// oscat_basic/POUs/List Processing/LIST_NEXT
FUNCTION_BLOCK LIST_NEXT
VAR_INPUT
	SEP : BYTE;
	RST : BOOL;
END_VAR
VAR_IN_OUT
	LIST : STRING(LIST_LENGTH);
END_VAR
VAR_OUTPUT
	LEL : STRING(LIST_LENGTH);
	NUL : BOOL;
END_VAR
VAR
	pos : INT := 1;
	pt : POINTER TO ARRAY[1..LIST_LENGTH] OF BYTE;
	po : POINTER TO ARRAY[1..LIST_LENGTH] OF BYTE;
	c: BYTE;
	write: INT;
END_VAR


(*
version 2.0	21. mar. 2011
programmer 	hugo
tested by		oscat

LIST_NEXT retrieves the next element of a list, starting from element 1 after reset or first init.
when the end of the lisat is reached a '' empty string is returned and NUL is set to true.
die liste liegt als string von elementen vor die mit den zeichen SEP am anfang markiert sind.

*)

pt := ADR(LIST);
po := ADR(LEL);

IF rst THEN
	pos := 1;
END_IF;

IF pt^[pos] = 0 OR pos = LIST_LENGTH THEN
	LEL := '';
	NUL := TRUE;
ELSE
	NUL := FALSE;
	write := 1;
	FOR pos := pos + 1 TO LIST_LENGTH DO
		c := pt^[pos];
		IF c = 0 OR c = SEP THEN
			po^[write] := 0;
			RETURN;
		ELSE
			po^[write] := pt^[pos];
			write := write + 1;
		END_IF;
	END_FOR;
END_IF;




(* revision histroy
hm	25. jun. 2008	rev 1.0
	original release

hm	19. jan. 2011	rev 1.1
	changed string(255) to string(LIST_LENGTH)	

hm	21. mar. 2011	rev 2.0
	all elements start with SEP

*)

END_FUNCTION_BLOCK

// oscat_basic/POUs/List Processing/LIST_RETRIEVE
FUNCTION LIST_RETRIEVE : STRING(LIST_LENGTH)
VAR_INPUT
	SEP : BYTE;
	POS : INT;
END_VAR

VAR
	i :	INT;
	o : INT := 1;
	w : INT := 1;
	pt : POINTER TO ARRAY[1..LIST_LENGTH] OF BYTE;
	po : POINTER TO ARRAY[1..LIST_LENGTH] OF BYTE;
	cnt: INT := 0;
	c: BYTE;
END_VAR


(*
version 2.0		21. mar. 2011
programmer 	hugo
tested by		oscat

LIST_RETRIEVE liefert das element an der stelle pos einer liste und löscht das element aus der liste.
die liste liegt als string von elementen vor die mit den zeichen SEP separiert sind.

*)
(*All VAR_IN_OUT variables have been moved to the end of the declaration due to compatibility reasons*)
VAR_IN_OUT
	LIST : STRING(LIST_LENGTH);
END_VAR

(* load pointers *)
pt := ADR(LIST);
po := ADR(LIST_RETRIEVE);

IF pos > 0 THEN
	FOR i := 1 TO LIST_LENGTH DO
		c := pt^[i];
		IF c = 0 THEN
			po^[o] := 0;
			IF cnt < pos THEN pt^[w + 1] := 0; ELSE pt^[w] := 0; END_IF;
			RETURN;
		ELSIF cnt = pos AND c <> SEP THEN				(* we have found the element *)
			po^[o] := pt^[i];
			o := o + 1;
		ELSIF cnt >= pos THEN
			pt^[w] := c;
			w := w + 1;
		ELSE
			w := i;
		END_IF;
		IF c = sep THEN cnt := cnt + 1; END_IF;
	END_FOR;
ELSE
	LIST_RETRIEVE := '';
END_IF;


(* revision histroy
hm	28. jun. 2008	rev 1.0
	original release

hm	19. jan. 2011	rev 1.1
	changed string(255) to string(LIST_LENGTH)

hm	21. mar. 2011	rev 2.0
	all elements start with SEP
*)

END_FUNCTION

// oscat_basic/POUs/List Processing/LIST_RETRIEVE_LAST
FUNCTION LIST_RETRIEVE_LAST : STRING(LIST_LENGTH)
VAR_INPUT
	SEP : BYTE;
END_VAR

VAR
	i :	INT;
	last : INT := 1;
	pt : POINTER TO ARRAY[1..LIST_LENGTH] OF BYTE;
	c: BYTE;
END_VAR


(*
version 2.0		21. mar. 2011
programmer 	hugo
tested by		oscat

LIST_RETRIEVE_LAST liefert das letzte element einer liste und löscht das element aus der liste.
die liste liegt als string von elementen vor die mit den zeichen SEP beginnen.

*)
(*All VAR_IN_OUT variables have been moved to the end of the declaration due to compatibility reasons*)
VAR_IN_OUT
	LIST : STRING(LIST_LENGTH);
END_VAR

(* load pointers *)
pt := ADR(LIST);

(* search position of last element *)
FOR i := 1 TO LIST_LENGTH DO
	c := pt^[i];
	IF c = 0 THEN
		EXIT;
	ELSIF C = SEP THEN
		last := i;
	END_IF;
END_FOR;
(* return last element of list *)
LIST_RETRIEVE_LAST := MID(LIST, LIST_LENGTH, last + 1);
(* terminate list at i *)
pt^[last] := 0;



(* revision histroy
hm	21. mar. 2011	rev 2.0
	new module
*)

END_FUNCTION

// oscat_basic/POUs/Logic/FF edge triggered/COUNT_BR
FUNCTION_BLOCK COUNT_BR
VAR_INPUT
	SET : BOOL;
	IN : BYTE;
	UP : BOOL;
	DN : BOOL;
	STEP : BYTE := 1;
	MX : BYTE := 255;
	RST : BOOL;
END_VAR
VAR_OUTPUT
	CNT : BYTE;
END_VAR
VAR
	last_up: BOOL;
	last_dn: BOOL;
END_VAR

(*
	version 1.0	16 jan 2008
	programmer 	hugo
	tested BY	tobias

Count_BR is a byte counter with independen up and dn inputs. the counter counts from 0 to mx and continues at 0 after is has reached mx
a step input sets the counters stepping width.

*)

IF rst THEN
	cnt := 0;
ELSIF set THEN
	cnt := LIMIT(0,in,mx);
ELSIF up AND NOT last_up THEN
	cnt := INT_TO_BYTE(INC(cnt,step,mx));
ELSIF dn AND NOT last_dn THEN
	cnt := INT_TO_BYTE(inc(cnt,-step,mx));
END_IF;
last_up := up;
last_dn := dn;

(* revision history
hm	16. jan 2008	rev 1.0
	original version

*)

END_FUNCTION_BLOCK

// oscat_basic/POUs/Logic/FF edge triggered/COUNT_DR
FUNCTION_BLOCK COUNT_DR
VAR_INPUT
	SET : BOOL;
	IN : DWORD;
	UP : BOOL;
	DN : BOOL;
	STEP : DWORD := 1;
	MX : DWORD := 16#FFFFFFFF;
	RST : BOOL;
END_VAR
VAR_OUTPUT
	CNT : DWORD;
END_VAR
VAR
	last_up: BOOL;
	last_dn: BOOL;
END_VAR

(*
	version 1.1	20. jan. 2011
	programmer 	hugo
	tested BY		tobias

Count_DR is a DWORD counter with independen up and dn inputs. the counter counts from 0 to mx and continues at 0 after is has reached mx
a step input sets the counters stepping width.

*)

IF rst THEN
	cnt := 0;
ELSIF set THEN
	cnt := LIMIT(0,in,mx);
ELSIF up AND NOT last_up THEN
	IF STEP > MX - CNT THEN
		CNT := CNT - MX + STEP - 1;
	ELSE
		CNT := CNT + STEP;
	END_IF;
ELSIF dn AND NOT last_dn THEN
	IF STEP > CNT THEN
		CNT := CNT - STEP + MX + 1;
	ELSE
		CNT := CNT - STEP;
	END_IF;
END_IF;
last_up := up;
last_dn := dn;

(* revision history
hm	12. jun 2008	rev 1.0
	original version

hm	20. jan. 2011	rev 1.1
	corrected init value of MX to 16#FFFFFFFF

*)

END_FUNCTION_BLOCK

// oscat_basic/POUs/Logic/FF edge triggered/FF_D2E
FUNCTION_BLOCK FF_D2E
VAR_INPUT
	D0 : BOOL;
	D1 : BOOL;
	CLK : BOOL;
	RST : BOOL;
END_VAR
VAR_OUTPUT
	Q0 : BOOL;
	Q1 : BOOL;
END_VAR
VAR
	edge : BOOL;
END_VAR

(*
version 1.3	14. mar. 2009
programmer 	hugo
tested by		oscat

dual D-type flip flop with reset and rising clock trigger

*)

IF rst THEN
	Q0 := FALSE;
	Q1 := FALSE;
ELSIF clk AND NOT edge THEN
	Q0 := D0;
	Q1 := D1;
END_IF;
edge := CLK;

(* revision history
hm	25. dec 2007	rev 1.0
	original version

hm	27. dec 2007	rev 1.1
	changed code for better performance

hm	30. oct. 200	rev 1.2
	deleted unnecessary init with 0

hm	14. mar. 2009	rev 1.3
	removed double assignments

*)

END_FUNCTION_BLOCK

// oscat_basic/POUs/Logic/FF edge triggered/FF_D4E
FUNCTION_BLOCK FF_D4E
VAR_INPUT
	D0 : BOOL;
	D1 : BOOL;
	D2 : BOOL;
	D3 : BOOL;
	CLK : BOOL;
	RST : BOOL;
END_VAR
VAR_OUTPUT
	Q0 : BOOL;
	Q1 : BOOL;
	Q2 : BOOL;
	Q3 : BOOL;
END_VAR
VAR
	edge : BOOL;
END_VAR


(*
version 1.3	14. mar. 2009
programmer 	hugo
tested by		oscat

quad D-type flip flop with reset and rising clock trigger

*)

IF rst THEN
	Q0 := FALSE;
	Q1 := FALSE;
	Q2 := FALSE;
	Q3 := FALSE;
ELSIF clk AND NOT edge THEN
	Q0 := D0;
	Q1 := D1;
	Q2 := D2;
	Q3 := D3;
END_IF;
edge := CLK;

(* revision history
hm	4. aug 2006	rev 1.0
	original version

hm	27. dec 2007	rev 1.1
	changed code for better performance

hm	30. oct. 200	rev 1.2
	deleted unnecessary init with 0

hm	14. mar. 2009	rev 1.3
	removed double assignments

*)

END_FUNCTION_BLOCK

// oscat_basic/POUs/Logic/FF edge triggered/FF_DRE
FUNCTION_BLOCK FF_DRE
VAR_INPUT
	SET : BOOL;
	D : BOOL;
	CLK : BOOL;
	RST : BOOL;
END_VAR
VAR_OUTPUT
	Q : BOOL;
END_VAR
VAR
	edge : BOOL;
END_VAR


(*
version 1.2	30. oct. 2008
programmer 	hugo
tested by	oscat

D-type flip flop with set, reset and rising clock trigger

*)

IF rst OR set THEN
	Q := NOT rst;
ELSIF clk AND NOT edge THEN
	Q := D;
END_IF;
edge := CLK;

(* revision history
hm	4. aug 2006		rev 1.0
	original version

hm	27. dec 2007	rev 1.1
	changed code for better performance

hm	30. oct. 2008	rev 1.2
	optimized performance
*)

END_FUNCTION_BLOCK

// oscat_basic/POUs/Logic/FF edge triggered/FF_JKE
FUNCTION_BLOCK FF_JKE
VAR_INPUT
	SET : BOOL;
	J : BOOL;
	CLK : BOOL;
	K : BOOL;
	RST : BOOL;
END_VAR
VAR_OUTPUT
	Q : BOOL;
END_VAR
VAR
	edge : BOOL;
END_VAR


(*
version 1.2	30. oct. 2008
programmer 	hugo
tested by	oscat

JK-type flip flop with set, reset and rising clock trigger
set and reset are asynchron while the FF is rising edge triggered
J=0 and K=0 and CLK >>> no action
J=1 and K=0 and CLK >>> output = 1
J=0 and K=1 and CLK >>> output = 0
J=1 and K=1 and CLK >>> toggle output


*)

IF rst OR set THEN
	Q := NOT rst;
ELSIF clk AND NOT edge THEN
	IF J XOR K THEN Q := J;
	ELSE Q := K XOR Q;
	END_IF;
END_IF;
edge := CLK;

(* revision history
hm	4. aug 2006		rev 1.0
	original version

hm	27. dec 2007	rev 1.1
	changed code for better performance

hm	30. oct. 2008	rev 1.2
	optimized performance
*)

END_FUNCTION_BLOCK

// oscat_basic/POUs/Logic/FF edge triggered/FF_RSE
FUNCTION_BLOCK FF_RSE
VAR_INPUT
	CS : BOOL;
	CR : BOOL;
	RST : BOOL;
END_VAR
VAR_OUTPUT
	Q : BOOL;
END_VAR
VAR
	es, er : BOOL;
END_VAR

(*
version 1.0	16. jul. 2008
programmer 	hugo
tested by	oscat

this is a rising edge triggered rs flip flop
a rising edge on CS sets Q = TRUE and a rising edge on CR sets Q = FALSE.
CR has priority over CS.

*)

IF rst THEN
	(* asynchronous reset *)
	Q := FALSE;
ELSIF CR AND NOT er THEN
	(* rising edge on CR *)
	Q := FALSE;
ELSIF CS AND NOT es THEN
	(* rising edge on CS *)
	Q := TRUE;
END_IF;

es := CS;
er := CR;

(* revision history

hm	16. jul. 2008	rev 1.0
	original version

*)

END_FUNCTION_BLOCK

// oscat_basic/POUs/Logic/FF edge triggered/SELECT_8
FUNCTION_BLOCK SELECT_8
VAR_INPUT
	E : BOOL;
	SET : BOOL;
	IN : BYTE;
	UP : BOOL;
	DN : BOOL;
	RST : BOOL;
END_VAR
VAR_OUTPUT
	Q0, Q1, Q2, Q3, Q4, Q5, Q6, Q7 : BOOL;
	STATE : INT;
END_VAR
VAR
	last_up: BOOL;
	last_dn : BOOL;
END_VAR

(*
	version 1.1	27. feb. 2009
	programmer 	hugo
	tested BY		oscat

select_8 selects one of 8 outputs at any time. the outputscan be selected by up or down keys and an independent anable switches all outouts off if set false


*)

IF rst THEN
	state := 0;
ELSIF set THEN
	state := IN;
ELSIF up AND NOT last_up THEN
	state := inc(state,1,7);
ELSIF dn AND NOT last_dn THEN
	state := inc(state,-1,7);
END_IF;
last_UP := UP;
last_DN := DN;

Q0 := FALSE;
Q1 := FALSE;
Q2 := FALSE;
Q3 := FALSE;
Q4 := FALSE;
Q5 := FALSE;
Q6 := FALSE;
Q7 := FALSE;

IF E THEN
	CASE state OF
		0: Q0 := TRUE;
		1: Q1 := TRUE;
		2: Q2 := TRUE;
		3: Q3 := TRUE;
		4: Q4 := TRUE;
		5: Q5 := TRUE;
		6: Q6 := TRUE;
		7: Q7 := TRUE;
	END_CASE;
END_IF;

(* revision history
hm	16. jan 2008	rev 1.0
	original version

hm	27. feb. 2009	rev 1.1
	renamed input en to e
*)

END_FUNCTION_BLOCK

// oscat_basic/POUs/Logic/FF edge triggered/SHR_4E
FUNCTION_BLOCK SHR_4E
VAR_INPUT
	SET : BOOL;
	D0: BOOL;
	CLK: BOOL;
	RST: BOOL;
END_VAR
VAR_OUTPUT
	Q0: BOOL;
	Q1: BOOL;
	Q2: BOOL;
	Q3: BOOL;
END_VAR
VAR
	trig : R_TRIG;
END_VAR

(*
version 1.1	25. oct. 2008
programmer 	hugo
tested by		tobias

4 bit shift register with reset

*)

(* trig.Q signals a rising edge on clk *)
trig(clk := clk);

IF set OR rst THEN
	Q0 := NOT rst;
	Q1 := Q0;
	Q2 := Q0;
	Q3 := Q0;
ELSIF trig.Q THEN
	Q3 := Q2;
	Q2 := Q1;
	Q1 := Q0;
	Q0 := D0;
END_IF;



(* revision history
hm	4. aug. 2006	rev 1.0
	original version

hm	25. oct. 2008	rev 1.1
	optimized code

*)

END_FUNCTION_BLOCK

// oscat_basic/POUs/Logic/FF edge triggered/SHR_4UDE
FUNCTION_BLOCK SHR_4UDE
VAR_INPUT
	SET : BOOL;
	D0: BOOL;
	D3: BOOL;
	CLK: BOOL;
	DN : BOOL;
	RST: BOOL;

END_VAR
VAR_OUTPUT
	Q0: BOOL;
	Q1: BOOL;
	Q2: BOOL;
	Q3: BOOL;
END_VAR
VAR
	trig : R_TRIG;
END_VAR

(*
version 1.2	14. mar. 2009
programmer 	hugo
tested by		tobias

4 bit shift register with reset up / down direction input

*)

(* trig.Q signals a rising edge on clk *)
trig(clk := clk);

IF set OR rst THEN
	Q0 := NOT RST;
	Q1 := Q0;
	Q2 := Q0;
	Q3 := Q0;
ELSIF trig.Q THEN
	IF dn THEN
		Q0 := Q1;
		Q1 := Q2;
		Q2 := Q3;
		Q3 := D3;
	ELSE
		Q3 := Q2;
		Q2 := Q1;
		Q1 := Q0;
		Q0 := D0;
	END_IF;
END_IF;



(* revision history
hm	4. aug. 2006	rev 1.0
	original version

hm	25. oct. 2008	rev 1.1
	optimized code

hm	14. mar. 2009	rev 1.2
	removed double assignments

*)

END_FUNCTION_BLOCK

// oscat_basic/POUs/Logic/FF edge triggered/SHR_8PLE
FUNCTION_BLOCK SHR_8PLE
VAR_INPUT
	Din : BOOL;
	Dload : BYTE;
	CLK: BOOL;
	UP: BOOL :=1;
	load : BOOL;
	RST: BOOL;
END_VAR
VAR_OUTPUT
	DOut: BOOL;
END_VAR
VAR
	edge : BOOL :=1;
	register : BYTE;
END_VAR

(*
version 1.0	4 aug 2006
programmer 	hugo
tested by	oscat

8 bit shift register with reset and parallel load
the register can shift up or down
it also has a serial input.
the Din input is on Bit0 for up shift and on bit 7 for down shift
the Dout output is on Bit7 for up shift and on bit 0 for down shift
paralle clock is performed clock synchron while a shift is performed first and then the register is reloaded


*)

(* flankenerkennung clk wird high und edge war high reset ist nicht aktiv und set ist nicht aktiv *)
IF CLK AND edge AND NOT rst THEN
	edge := FALSE;	(* flanke wurde erkannt und weitere flankenerkennung wird verhindert bis edge wieder true ist *)
	(* hier ist der code für das flankenevent *)
	IF UP THEN						(*shift up *)
		register := SHL(register,1);
		register.0 := Din;
		Dout := register.7;
	ELSE								(* shift down *);
		register := SHR(register,1);
		register.7 := Din;
		Dout := register.0;
	END_IF;
	IF load THEN							(* the byte on Din will be loaded if load = true *)
		register := Dload;
		IF up THEN Dout := register.7; ELSE Dout := register.0; END_IF;
	END_IF;
END_IF;
IF NOT clk THEN edge := TRUE; END_IF;	(* sobald clk wieder low wird warten auf nächste flanke *)
IF rst THEN									(* wenn reset aktiv dann ausgang rücksetzen *)
	register := 0;
	Dout := FALSE;
END_IF;

END_FUNCTION_BLOCK

// oscat_basic/POUs/Logic/FF edge triggered/SHR_8UDE
FUNCTION_BLOCK SHR_8UDE
VAR_INPUT
	SET : BOOL;
	D0: BOOL;
	D7: BOOL;
	CLK: BOOL;
	DN : BOOL;
	RST: BOOL;
END_VAR
VAR_OUTPUT
	Q0: BOOL;
	Q1: BOOL;
	Q2: BOOL;
	Q3: BOOL;
	Q4: BOOL;
	Q5: BOOL;
	Q6: BOOL;
	Q7: BOOL;
END_VAR
VAR
	trig : R_TRIG;
END_VAR

(*
version 1.2	14. mar. 2009
programmer 	hugo
tested by		tobias

8 bit shift register with reset


*)

(* trig.Q signals a rising edge on clk *)
trig(clk := clk);

IF set OR rst THEN
	Q0 := NOT RST;
	Q1 := Q0;
	Q2 := Q0;
	Q3 := Q0;
	Q4 := Q0;
	Q5 := Q0;
	Q6 := Q0;
	Q7 := Q0;
ELSIF trig.Q THEN
	IF dn THEN
		Q0 := Q1;
		Q1 := Q2;
		Q2 := Q3;
		Q3 := Q4;
		Q4 := Q5;
		Q5 := Q6;
		Q6 := Q7;
		Q7 := D7;
	ELSE
		Q7 := Q6;
		Q6 := Q5;
		Q5 := Q4;
		Q4 := Q3;
		Q3 := Q2;
		Q2 := Q1;
		Q1 := Q0;
		Q0 := D0;
	END_IF;
END_IF;



(* revision history
hm	4. aug. 2006	rev 1.0
	original version

hm	25. oct. 2008	rev 1.1
	optimized code

hm	14. mar. 2009	rev 1.2
	removed double assignments

*)

END_FUNCTION_BLOCK

// oscat_basic/POUs/Logic/FF pulse triggered/LTCH
FUNCTION_BLOCK LTCH
VAR_INPUT
	D : BOOL;
	L : BOOL;
	RST : BOOL;
END_VAR
VAR_OUTPUT
	Q : BOOL;
END_VAR


(*
version 1.2	30. oct. 2008
programmer 	hugo
tested by	oscat

Transparent Latch with asynchronous reset


*)

(* as long as L is true, the latch is transparent and and change of D is transferred to Q *)
(* of course only when there is no asynchronous reset *)
IF rst THEN				(* if asynchronous reset then Q=0 *)
	Q := FALSE;
ELSIF L THEN			(* latch is transparent *)
	Q := D;
END_IF;


(* revision history
hm	4. aug 2006		rev 1.0
	original version

hm	27. dec 2007	rev 1.1
	changed code for better performance

hm	30. oct. 2008	rev 1.2
	deleted unnecessary init with 0

*)

END_FUNCTION_BLOCK

// oscat_basic/POUs/Logic/FF pulse triggered/LTCH_4
FUNCTION_BLOCK LTCH_4
VAR_INPUT
	D0 : BOOL;
	D1 : BOOL;
	D2 : BOOL;
	D3 : BOOL;
	L : BOOL;
	RST : BOOL;
END_VAR
VAR_OUTPUT
	Q0 : BOOL;
	Q1 : BOOL;
	Q2 : BOOL;
	Q3 : BOOL;
END_VAR


(*
version 1.3	14. mar. 2009
programmer 	hugo
tested by		oscat

Quad Transparent Latch with asynchronous reset


*)

(* as long as L is true, the latch is transparent and and change of D is transferred to Q *)
(* of course only when there is no asynchronous reset *)
IF rst THEN			(* if asynchronous reset then Q=0 *)
	Q0 := FALSE;
	Q1 := FALSE;
	Q2 := FALSE;
	Q3 := FALSE;
ELSIF L THEN			(* latch is transparent *)
	Q0 := D0;
	Q1 := D1;
	Q2 := D2;
	Q3 := D3;
END_IF;

(* revision history
hm	4. aug 2006	rev 1.0
	original version

hm	27. dec 2007	rev 1.1
	changed code for better performance

hm	30. oct. 2008	rev 1.2
	deleted unnecessary init with 0

hm	14. mar. 2009	rev 1.3
	removed double assignments

*)

END_FUNCTION_BLOCK

// oscat_basic/POUs/Logic/FF pulse triggered/STORE_8
FUNCTION_BLOCK STORE_8
VAR_INPUT
	Set : BOOL;
	D0,D1, D2, D3, D4, D5, D6, D7 : BOOL;
	Clr : BOOL;
	Rst : BOOL;
END_VAR
VAR_OUTPUT
	Q0, Q1, Q2, Q3, Q4, Q5, Q6, Q7 : BOOL;
END_VAR
VAR
	edge: BOOL;
END_VAR

(*
version 1.2	14. mar. 2009
programmer 	hugo
tested by		oscat

Store_4 stores up to 4 boolean inputs until a reset is clearing the outputs.
the respective output is set with a true at the respective input and stays true until a reset is generated.
a set input is used to set all outputs true at the same time, independent of their inputs.
a clear input is used to reset only the lowest priority of the outputs one at a time.
the lowest priority is q3.

*)

IF rst OR set THEN
	q0 := NOT rst;
	q1 := q0;
	q2 := q0;
	q3 := q0;
	q4 := q0;
	q5 := q0;
	q6 := q0;
	q7 := q0;
ELSE
	IF D0 THEN Q0 := TRUE; END_IF;
	IF D1 THEN Q1 := TRUE; END_IF;
	IF D2 THEN Q2 := TRUE; END_IF;
	IF D3 THEN Q3 := TRUE; END_IF;
	IF D4 THEN Q4 := TRUE; END_IF;
	IF D5 THEN Q5 := TRUE; END_IF;
	IF D6 THEN Q6 := TRUE; END_IF;
	IF D7 THEN Q7 := TRUE; END_IF;

	IF clr AND NOT edge THEN
		IF q0 THEN q0 := FALSE;
		ELSIF q1 THEN q1 := FALSE;
		ELSIF q2 THEN q2 := FALSE;
		ELSIF q3 THEN q3 := FALSE;
		ELSIF q4 THEN q4 := FALSE;
		ELSIF q5 THEN q5 := FALSE;
		ELSIF q6 THEN q6 := FALSE;
		ELSE q7 := FALSE;
		END_IF;
	END_IF;
	edge := clr;
END_IF;


(* revision history
hm	25.12.2007	rev 1.0
	original version

hm	30. oct. 2008	rev 1.1
	optimized performance

hm	14. mar. 2009	rev 1.2
	removed double assignments

*)

END_FUNCTION_BLOCK

// oscat_basic/POUs/Logic/gate logic/BCDC_TO_INT
FUNCTION BCDC_TO_INT : INT
VAR_INPUT
	IN : BYTE;
END_VAR


(*
version 1.1 30. jun. 2008
programmer 	hugo
tested by	oscat

this function converts a two digit bcd number into an integer.

*)

BCDC_TO_INT := (in AND 16#0F) + (SHR(in,4) * 10);

(* revision history
hm	13.12.2007	rev 1.0
	original version

hm	30.6.2008	rev 1.1
	changed name BCD_TO_INT to BCDC_TO_INT to avoid collision with util.lib

*)

END_FUNCTION

// oscat_basic/POUs/Logic/gate logic/BIT_LOAD_B
FUNCTION BIT_LOAD_B : BYTE
VAR_INPUT
	IN : BYTE;
	VAL : BOOL;
	POS : INT;
END_VAR
VAR CONSTANT
	dat : BYTE := 1;
END_VAR

(*
version 1.1	16. mar 2008
programmer 	hugo
tested by	tobias

this function loads a bit into a byte at position pos.
 *)

IF VAL THEN
	BIT_LOAD_B := in OR SHL(dat,pos);
ELSE
	BIT_LOAD_B := in AND (NOT SHL(dat,pos));
END_IF;


(* revision history
hm	29. feb 2008	rev 1.0
	original version

hm	16. mar 2008	rev 1.1
	change input bit to val for compatibility reasons
*)

END_FUNCTION

// oscat_basic/POUs/Logic/gate logic/BIT_LOAD_B2
FUNCTION BIT_LOAD_B2 : BYTE
VAR_INPUT
	I : BYTE;
	D : BOOL;
	P : INT;
	N : INT;
END_VAR


(*
version 1.0 18. oct. 2008
programmer 	hugo
tested by	tobias

this function loads N bits of D at pos P in Byte I

*)

IF D THEN
	BIT_LOAD_B2 := ROL(SHR(BYTE#255, 8 - N) OR ROR(i, P), P);
ELSE
	BIT_LOAD_B2 := ROL(SHL(BYTE#255, N) AND ROR(I, P), P);
END_IF;



(* revision history
hm	18. oct. 2008	rev 1.0
	original version


*)

END_FUNCTION

// oscat_basic/POUs/Logic/gate logic/BIT_LOAD_DW
FUNCTION BIT_LOAD_DW : DWORD
VAR_INPUT
	IN : DWORD;
	VAL : BOOL;
	POS : INT;
END_VAR
VAR CONSTANT
	dat : DWORD := 1;
END_VAR

(*
version 1.1	16. mar 2008
programmer 	hugo
tested by	tobias

this function loads a bit into a DWord at position pos.
 *)

IF val THEN
	BIT_LOAD_DW := in OR SHL(dat,pos);
ELSE
	BIT_LOAD_DW := in AND (NOT SHL(dat,pos));
END_IF;


(* revision history
hm	29. feb 2008	rev 1.0
	original version

hm	16. mar 2008	rev 1.1
	change input bit to val for compatibility reasons
*)

END_FUNCTION

// oscat_basic/POUs/Logic/gate logic/BIT_LOAD_DW2
FUNCTION BIT_LOAD_DW2 : DWORD
VAR_INPUT
	I : DWORD;
	D : BOOL;
	P : INT;
	N : INT;
END_VAR


(*
version 1.0 18. oct. 2008
programmer 	hugo
tested by	tobias

this function loads N bits of D at pos P in DWORD I

*)

IF D THEN
	BIT_LOAD_DW2 := ROL(SHR(DWORD#4294967295, 32 - N) OR ROR(i, P), P);
ELSE
	BIT_LOAD_DW2 := ROL(SHL(DWORD#4294967295, N) AND ROR(I, P), P);
END_IF;



(* revision history
hm	18. oct. 2008	rev 1.0
	original version


*)

END_FUNCTION

// oscat_basic/POUs/Logic/gate logic/BIT_LOAD_W
FUNCTION BIT_LOAD_W : WORD
VAR_INPUT
	IN : WORD;
	VAL : BOOL;
	POS : INT;
END_VAR
VAR CONSTANT
	dat : WORD := 1;
END_VAR

(*
version 1.1	16. mar 2008
programmer 	hugo
tested by	tobias

this function loads a bit into a Word at position pos.
 *)

IF val THEN
	BIT_LOAD_W := in OR SHL(dat,pos);
ELSE
	BIT_LOAD_W := in AND (NOT SHL(dat,pos));
END_IF;


(* revision history
hm	29. feb 2008	rev 1.0
	original version

hm	16. mar 2008	rev 1.1
	change input bit to val for compatibility reasons
*)

END_FUNCTION

// oscat_basic/POUs/Logic/gate logic/BIT_LOAD_W2
FUNCTION BIT_LOAD_W2 : WORD
VAR_INPUT
	I : WORD;
	D : BOOL;
	P : INT;
	N : INT;
END_VAR


(*
version 1.0 18. oct. 2008
programmer 	hugo
tested by	tobias

this function loads N bits of D at pos P in WORD I

*)

IF D THEN
	BIT_LOAD_W2 := ROL(SHR(WORD#65535, 16 - N) OR ROR(i, P), P);
ELSE
	BIT_LOAD_W2 := ROL(SHL(WORD#65535, N) AND ROR(I, P), P);
END_IF;



(* revision history
hm	18. oct. 2008	rev 1.0
	original version


*)

END_FUNCTION

// oscat_basic/POUs/Logic/gate logic/BIT_OF_DWORD
FUNCTION BIT_OF_DWORD : BOOL
VAR_INPUT
	in : DWORD;
	N : INT;
END_VAR


(*
version 1.2	6. jun. 2008
programmer 	hugo
tested by	tobias

this function extracts a single bit from the nth position from right (right is lowest bit)
the lowest Bit (Bit0 from in) is selected with N=0.
 *)

BIT_OF_DWORD := (SHR(in,N) AND 16#00000001) > 0;


(* old code used before rev 1.1
temp := SHR(in,n);
Bit_of_Dword := temp.0;
*)


(* revision history
hm	4. aug. 2006	rev 1.0
	original version

hm	29. feb 2008	rev 1.1
	improved performance

hm	6. jun. 2008	rev 1.2
	changes type of input N from byte to int
*)

END_FUNCTION

// oscat_basic/POUs/Logic/gate logic/BIT_TOGGLE_B
FUNCTION BIT_TOGGLE_B : BYTE
VAR_INPUT
	IN : BYTE;
	POS : INT;
END_VAR


(*
version 1.0 18. oct. 2008
programmer 	hugo
tested by	tobias

this function toggles a bit of a BYTE at position pos.

*)

BIT_TOGGLE_B := SHL(BYTE#1, POS) XOR IN;




(* revision history
hm	18. oct. 2008	rev 1.0
	original version


*)

END_FUNCTION

// oscat_basic/POUs/Logic/gate logic/BIT_TOGGLE_DW
FUNCTION BIT_TOGGLE_DW : DWORD
VAR_INPUT
	IN : DWORD;
	POS : INT;
END_VAR


(*
version 1.0 18. oct. 2008
programmer 	hugo
tested by	tobias

this function toggles a bit of a WORD at position pos.

*)

BIT_TOGGLE_DW := SHL(DWORD#1, POS) XOR IN;



(* revision history
hm	18. oct. 2008	rev 1.0
	original version


*)

END_FUNCTION

// oscat_basic/POUs/Logic/gate logic/BIT_TOGGLE_W
FUNCTION BIT_TOGGLE_W : WORD
VAR_INPUT
	IN : WORD;
	POS : INT;
END_VAR


(*
version 1.0 18. oct. 2008
programmer 	hugo
tested by	tobias

this function toggles a bit of a WORD at position pos.

*)

BIT_TOGGLE_W := SHL(WORD#1, POS) XOR IN;



(* revision history
hm	18. oct. 2008	rev 1.0
	original version


*)

END_FUNCTION

// oscat_basic/POUs/Logic/gate logic/BYTE_OF_BIT
FUNCTION BYTE_OF_BIT : BYTE
VAR_INPUT
	B0:BOOL;
	B1:BOOL;
	B2:BOOL;
	B3:BOOL;
	B4:BOOL;
	B5:BOOL;
	B6:BOOL;
	B7:BOOL;
END_VAR


(*
version 1.1	 18. feb 2006
programmer 	hugo
tested by		tobias

this function creates a byte from 8 individual bits

*)

Byte_of_bit := SHL(SHL(SHL(SHL(SHL(SHL(SHL(BOOL_TO_BYTE(B7),1) OR BOOL_TO_BYTE(B6),1) OR BOOL_TO_BYTE(B5),1) OR BOOL_TO_BYTE(B4),1)
	OR BOOL_TO_BYTE(B3),1) OR BOOL_TO_BYTE(B2),1) OR BOOL_TO_BYTE(B1),1) OR BOOL_TO_BYTE(B0);


(* revision history

hm	4. aug 2006		rev 1.0
	original version

hm	18. feb. 2008	rev 1.1
	improved performance

*)

END_FUNCTION

// oscat_basic/POUs/Logic/gate logic/BYTE_OF_DWORD
FUNCTION BYTE_OF_DWORD : BYTE
VAR_INPUT
	in : DWORD;
	N : BYTE;
END_VAR


(*
version 1.2	30. oct. 2008
programmer 	hugo
tested by	oscat

this function extracts a single byte from the nth position from right (right is lowest byte) 
the lower byte (starting with Bit0 from in) is selected with N=0.
*)

BYTE_OF_DWORD := DWORD_TO_BYTE(SHR(in,SHL(n,3)));

(* revision history
hm	17. jan 2007	rev 1.0
	original version

hm	2. jan 2008		rev 1.1
	improved performance

hm	30. oct. 2008	rev 1.2
	improved performance
*)

END_FUNCTION

// oscat_basic/POUs/Logic/gate logic/BYTE_TO_BITS
FUNCTION_BLOCK BYTE_TO_BITS
VAR_INPUT
	IN: BYTE;
END_VAR
VAR_OUTPUT
	B0: BOOL;
	B1: BOOL;
	B2: BOOL;
	B3: BOOL;
	B4: BOOL;
	B5: BOOL;
	B6: BOOL;
	B7: BOOL;
END_VAR


(*
version 1.1	16. mar. 2008
programmer 	hugo
tested by		tobias

this Function Block extracts the 8 Bits from a byte


*)

B0 := IN.0;
B1 := IN.1;
B2 := IN.2;
B3 := IN.3;
B4 := IN.4;
B5 := IN.5;
B6 := IN.6;
B7 := IN.7;

(* revision history
hm		4. aug 2006	rev 1.0
	original version

hm		16. mar 2008	rev 1.1
	renamed from byte_to_bit to byte_to_bits for compatibility reasons

*)

END_FUNCTION_BLOCK

// oscat_basic/POUs/Logic/gate logic/BYTE_TO_GRAY
FUNCTION BYTE_TO_GRAY : BYTE
VAR_INPUT
	IN : BYTE;
END_VAR


(*
version 1.0	9. nov. 2009
programmer 	hugo
tested by		oscat

this function converts a binary to gray code

*)

BYTE_TO_GRAY := IN XOR SHR(IN,1);

(* revision history
hm	9. nov. 2009	rev 1.0
	original version

*)

END_FUNCTION

// oscat_basic/POUs/Logic/gate logic/CHECK_PARITY
FUNCTION CHECK_PARITY : BOOL
VAR_INPUT
	in : DWORD;
	p : BOOL;
END_VAR


(*
version 1.3	18 feb 2008
programmer 	hugo
tested by	tobias

this function checks for an even partity for a dword and partity bit.

*)

CHECK_PARITY := NOT p;
WHILE in > 0 DO
	CHECK_PARITY := CHECK_PARITY XOR in.0 XOR in.1 XOR in.2 XOR in.3;
	in := SHR(in,4);
END_WHILE;

(* code before rev 1.2
WHILE in > 0 DO
	IF in.0 THEN cnt := cnt + 1; END_IF;
	in := SHR(in,1);
END_WHILE;
check_parity := even(cnt) XOR P;
*)


(* revision history

rev 1.0 HM  1.oct.2006

rev 1.1 hm	10.sep.2007
	changed algorithm to improove performance

rev 1.2	hm	8 dec 2007
	changed algorithm to improove performance

rev 1.3 hm	18. feb 2008
	changed algorithm to improove performance
*)

END_FUNCTION

// oscat_basic/POUs/Logic/gate logic/CHK_REAL
FUNCTION CHK_REAL : BYTE
VAR_INPUT
	X : REAL;
END_VAR
VAR
	pt : POINTER TO DWORD;
	tmp : DWORD;
END_VAR


(*
version 1.0	20. jan. 2011
programmer 	hugo
tested by		tobias

this function checks a floating point variable of type real (IEEE754-32Bits) for NAN and infinity
RETURN values: #0 = normal value, #20 = +infinity, #40 = -infinty, #80 = NAN

*)

pt := ADR(X);				(* move real to dword, real_to_dword does not work becasze it treats dword as a number on many systems *)
tmp := ROL(pt^,1);			(* rotate left foir easy checking, sign will be at lease significant digit *)
IF tmp < 16#FF000000 THEN
	CHK_REAL := 16#00;		(* normalized and denormalized numbers *)
ELSIF tmp = 16#FF000000 THEN
	CHK_REAL := 16#20;		(* X is +infinity see IEEE754 *)
ELSIF tmp = 16#FF000001 THEN
	CHK_REAL := 16#40;		(* X is -infinity see IEEE754 *)
ELSE
	CHK_REAL := 16#80;		(* X is NAN see IEEE754 *)
END_IF;


(* revision history
hm	 20. jan. 2011	rev 1.0
	original version

*)

END_FUNCTION

// oscat_basic/POUs/Logic/gate logic/DEC_2
FUNCTION_BLOCK DEC_2
VAR_INPUT
	D: BOOL;
	A: BOOL;
END_VAR
VAR_OUTPUT
	Q0: BOOL;
	Q1: BOOL;
END_VAR


(*
version 1.1	3 Mar 2007
programmer 	hugo
tested by		tobias

a bit input will be decoded to the two outputs Q0 or Q1
dependent on the value of A
A=0 decodes to Q0 and A=1 decodes to Q1

*)

Q0 := D AND NOT A;
Q1 := D AND A;

(* revision history
hm 3.3.2007	rev 1.1
	rewritten in ST for better compatibility

*)

END_FUNCTION_BLOCK

// oscat_basic/POUs/Logic/gate logic/DEC_4
FUNCTION_BLOCK DEC_4
VAR_INPUT
	D: BOOL;
	A0: BOOL;
	A1: BOOL;
END_VAR
VAR_OUTPUT
	Q0: BOOL;
	Q1: BOOL;
	Q2: BOOL;
	Q3: BOOL;
END_VAR


(*
version 1.1	3 Mar 2007
programmer 	hugo
tested by		tobias

a bit input will be decoded to one of the 4 outputs
dependent on the Adress on A0 and A1

executioin TIME on wago 750-841 = 9us
*)

Q0 := D AND NOT A0 AND NOT A1;
Q1 := D AND A0 AND NOT A1;
Q2 := D AND NOT A0 AND A1;
Q3 := D AND A0 AND A1;

(* revision history
hm 3.3.2007	rev 1.1
	rewritten in ST for better compatibility

*)

END_FUNCTION_BLOCK

// oscat_basic/POUs/Logic/gate logic/DEC_8
FUNCTION_BLOCK DEC_8
VAR_INPUT
	D: BOOL;
	A0: BOOL;
	A1: BOOL;
	A2: BOOL;
END_VAR
VAR_OUTPUT
	Q0: BOOL;
	Q1: BOOL;
	Q2: BOOL;
	Q3: BOOL;
	Q4: BOOL;
	Q5: BOOL;
	Q6: BOOL;
	Q7: BOOL;
END_VAR
VAR
	X : INT;
END_VAR

(*
version 1.3	28. mar. 2009
programmer 	hugo
tested by		oscat

a bit input will be decoded to one of the 8 outputs
dependent on the Adress on A0, A1 and A2


*)

X.0 := A0; X.1 := A1; X.2 := A2;

Q0 := FALSE;
Q1 := FALSE;
Q2 := FALSE;
Q3 := FALSE;
Q4 := FALSE;
Q5 := FALSE;
Q6 := FALSE;
Q7 := FALSE;

CASE X OF
	0 : Q0 := D;
	1 : Q1 := D;
	2 : Q2 := D;
	3 : Q3 := D;
	4 : Q4 := D;
	5 : Q5 := D;
	6 : Q6 := D;
	7 : Q7 := D;
END_CASE;



(* revision history
hm 3. mar. 2007	rev 1.1
	rewritten in ST for better compatibility

hm	26. oct. 2008	rev 1.2
	code optimized

hm	28. mar. 2009	rev 1.3
	replaced multiple assignments
*)

END_FUNCTION_BLOCK

// oscat_basic/POUs/Logic/gate logic/DW_TO_REAL
FUNCTION DW_TO_REAL : REAL
VAR_INPUT
	X : DWORD;
END_VAR
VAR
	pt : POINTER TO REAL;
END_VAR

(*
version 1.0	18. apr. 2008
programmer 	hugo
tested by		tobias

this function converts a DWORD to REAL in a bitwise manner.
*)

pt := ADR(X);
DW_TO_REAL := pt^;

(* revision history
hm	18. apr. 2008
	original version

*)

END_FUNCTION

// oscat_basic/POUs/Logic/gate logic/DWORD_OF_BYTE
FUNCTION DWORD_OF_BYTE : DWORD
VAR_INPUT
	B3 : BYTE;
	B2 : BYTE;
	B1 : BYTE;
	B0 : BYTE;
END_VAR


(*
version 1.3	18. jul. 2009
programmer 	hugo
tested by		tobias

this function creates a Dword from 4 individual bytes

*)

DWORD_OF_BYTE := SHL(SHL(SHL(BYTE_TO_DWORD(B3),8) OR BYTE_TO_DWORD(B2),8) OR BYTE_TO_DWORD(B1),8) OR BYTE_TO_DWORD(B0);


(* revision history
hm	24. jan 2007	rev 1.0
	original version

hm 2. jan 2008	rev 1.1
	inproved performance

hm	23. apr. 2008	rev 1.2
	reverse order of inputs to be more logical

hm	18. jul. 2009	rev 1.3
	added type conversions for compatibility reasons
*)

END_FUNCTION

// oscat_basic/POUs/Logic/gate logic/DWORD_OF_WORD
FUNCTION DWORD_OF_WORD : DWORD
VAR_INPUT
	W1 : WORD;
	W0 : WORD;
END_VAR


(*
version 1.0	18. jul. 2009
programmer 	hugo
tested by		tobias

this function creates a Dword from 2 individual Words

*)

DWORD_OF_WORD := SHL(WORD_TO_DWORD(W1),16) OR WORD_TO_DWORD(W0);


(* revision history

hm	18. jul. 2009	rev 1.0
	original version

*)

END_FUNCTION

// oscat_basic/POUs/Logic/gate logic/GRAY_TO_BYTE
FUNCTION GRAY_TO_BYTE : BYTE
VAR_INPUT
	IN : BYTE;
END_VAR


(*
version 1.0	9. nov. 2009
programmer 	hugo
tested by		oscat

this function converts a gray code into binary

*)

GRAY_TO_BYTE := SHR(IN,4) XOR IN;
GRAY_TO_BYTE := SHR(GRAY_TO_BYTE,2) XOR GRAY_TO_BYTE;
GRAY_TO_BYTE := SHR(GRAY_TO_BYTE,1) XOR GRAY_TO_BYTE;

(* revision history
hm	9. nov. 2009	rev 1.0
	original version

*)

END_FUNCTION

// oscat_basic/POUs/Logic/gate logic/INT_TO_BCDC
FUNCTION INT_TO_BCDC : BYTE
VAR_INPUT
	IN : INT;
END_VAR


(*
version 1.1	30. jun. 2008
programmer 	hugo
tested by		tobias

this function converts an integer into a two digit bcd number.
*)

INT_TO_BCDC := SHL(INT_TO_BYTE(IN / INT#10),4) OR INT_TO_BYTE(in MOD INT#10);

(* revision history
hm	13.12.2007
	original version

hm	30.6.2008	rev 1.1
	changed name INT_TO_BCD to INT_TO_BCDC to avoid collision with util.lib
	corrected error in code

*)

END_FUNCTION

// oscat_basic/POUs/Logic/gate logic/MUX_2
FUNCTION MUX_2 : BOOL
VAR_INPUT
	D0: BOOL;
	D1: BOOL;
	A0: BOOL;
END_VAR


(*
	version 1.2	16. oct. 2008
	programmer 	hugo
	tested BY	oscat

	dual input multiplexer
	depending on the value of A0, D0 or D1 will be switched to the Output

	executioin TIME on wago 750-841 = 7us
*)

MUX_2 := SEL(A0, D0, D1);


(*
revision history:
hm	5.10.2006		rev 1.1
	changed to ST Langage for better portability.

hm	16. oct. 2008	rev 1.2
	improved performance

*)

END_FUNCTION

// oscat_basic/POUs/Logic/gate logic/MUX_4
FUNCTION MUX_4 : BOOL
VAR_INPUT
	D0: BOOL;
	D1: BOOL;
	D2: BOOL;
	D3: BOOL;
	A0: BOOL;
	A1: BOOL;
END_VAR


(*
version 1.2	16. oct. 2008
programmer 	hugo
tested BY	oscat

quad input multiplexer
depending on the value of A0 and A1, one of the 4 inputs will be switched to the Output


*)

IF A1 THEN
	MUX_4 := SEL(A0, D2, D3);
ELSE
	MUX_4 := SEL(A0, D0, D1);
END_IF;


(*
revision history:
hm 	5.10.2006		rev 1.1
	rewritten to ST for better portability

hm	16. oct. 2008	rev 1.2
	improved performance

*)

END_FUNCTION

// oscat_basic/POUs/Logic/gate logic/PARITY
FUNCTION PARITY : BOOL
VAR_INPUT
	in : DWORD;
END_VAR


(*
	version 1.3	18 feb 2008
	programmer 	hugo
	tested BY		hans

this function calculates the even parity of an input Dword
the output will be true if the amount of high bits are an odd number.

*)

WHILE in > 0 DO
	PARITY := PARITY XOR in.0 XOR in.1 XOR in.2 XOR in.3;
	in := SHR(in,4);
END_WHILE;

(* code before rev 1.2
WHILE in > 0 DO
	IF in.0 THEN cnt := cnt +1; END_IF;
	in := SHR(in,1);
END_WHILE;
IF (cnt MOD 2) = 1 THEN parity := TRUE; ELSE parity := FALSE; END_IF;
*)

(* revision history

rev 1.0 hm 1 sep 2006
	original version

rev 1.1 hm 10.9.2007
	changed algorithm to improve performance

rev 1.2	hm	8 dec 2007
	changed algorithm to improve performance

rev 1.3	hm	18 feb 2008
	changed algorithm to improve performance
*)

END_FUNCTION

// oscat_basic/POUs/Logic/gate logic/REAL_TO_DW
FUNCTION REAL_TO_DW : DWORD
VAR_INPUT
	X : REAL;
END_VAR
VAR
	pt : POINTER TO DWORD;
END_VAR

(*
version 1.0	18. apr. 2008
programmer 	hugo
tested by		tobias

this function converts a 32 Bit Real to a dword in a bitwise manner.
*)

pt := ADR(X);
REAL_TO_DW := pt^;

(* revision history
hm	18. apr. 2008
	original version

*)

END_FUNCTION

// oscat_basic/POUs/Logic/gate logic/REFLECT
FUNCTION REFLECT : DWORD
VAR_INPUT
	D : DWORD;
	L : INT;
END_VAR
VAR
	i : INT;
END_VAR


(*
	version 1.0	16. jan 2011
	programmer 	hugo
	tested BY		tobias

This function reverses the specified amount of bits from bit 0 to bit n within a dword  while L specifies the amount of Bits to be reflected.

*)

REFLECT := 0;
FOR i := 1 TO L DO
	REFLECT := SHL(REFLECT, 1) OR BOOL_TO_DWORD(D.0);
	D := SHR(D, 1);
END_FOR;
REFLECT := REFLECT OR SHL(D, L);

(* revision history
hm	 16. jan 2011
	new module

*)

END_FUNCTION

// oscat_basic/POUs/Logic/gate logic/SHL1
FUNCTION SHL1 : DWORD
VAR_INPUT
	IN : DWORD;
	N : INT;
END_VAR
VAR CONSTANT
	temp : DWORD := 16#FFFF_FFFF;
END_VAR

(*
version 1.1	27 dec 2007
programmer 	hugo
tested by		tobias

SHL1 shifts N bits to the left filling the new bits with 1

*)

SHL1 := SHR(temp,32-N) OR SHL(IN,N);


(* revision history
hm	14.9.2007		rev 1.0
	original version

hm	27. dec 2007	rev 1.1
	changed code for better performance

*)

END_FUNCTION

// oscat_basic/POUs/Logic/gate logic/SHR1
FUNCTION SHR1 : DWORD
VAR_INPUT
	IN : DWORD;
	N : INT;
END_VAR
VAR CONSTANT
	temp : DWORD := 16#FFFF_FFFF;
END_VAR

(*
version 1.1	27 dec 2007
programmer 	hugo
tested by		tobias

SHR1 shifts N bits to the right filling the new bits with 1

*)

SHR1 := SHL(temp,32-N) OR SHR(IN,N);

(* revision history
hm	14.9.2007		rev 1.0
	original version

hm	27. dec 2007	rev 1.1
	changed code for better performance

*)

END_FUNCTION

// oscat_basic/POUs/Logic/gate logic/SWAP_BYTE
FUNCTION SWAP_BYTE : WORD
VAR_INPUT
	IN : WORD;
END_VAR


(*
version 1.0	4 feb 2008
programmer 	hugo
tested by		tobias

This function swaps the high and low byte of the word in.

*)

SWAP_BYTE := ROL(in,8);


(* revision history
hm		4. feb 2008	rev 1.0
	original version

*)

END_FUNCTION

// oscat_basic/POUs/Logic/gate logic/SWAP_BYTE2
FUNCTION SWAP_BYTE2 : DWORD
VAR_INPUT
	IN : DWORD;
END_VAR


(*
version 1.0	4 feb 2008
programmer 	hugo
tested by		tobias

This function reverses the byte order in the dword.

*)

Swap_Byte2 := (ROR(in,8) AND 16#FF00FF00) OR (ROL(in,8) AND 16#00FF00FF);

(* revision history
hm		4. feb 2008	rev 1.0
	original version

*)

END_FUNCTION

// oscat_basic/POUs/Logic/gate logic/WORD_OF_BYTE
FUNCTION WORD_OF_BYTE : WORD
VAR_INPUT
	B1 : BYTE;
	B0 : BYTE;
END_VAR


(*
version 1.4	18. jul. 2009
programmer 	hugo
tested by		tobias

this function creates a word from 2 individual bytes

*)

WORD_OF_BYTE := SHL(BYTE_TO_WORD(B1),8) OR BYTE_TO_WORD(B0);

(* revision history
hm	24. jan 2007	rev 1.0
	original version

hm	2. jan 2008	rev 1.1
	improved performance

hm	19. feb 2008	rev 1.2
	replaced and with or for better compatibility

hm	23. apr. 2008	rev 1.3
	reverse order of inputs to be more logical

hm	18. jul. 2009	rev 1.4
	added type conversions for compatibility reasons

*)

END_FUNCTION

// oscat_basic/POUs/Logic/gate logic/WORD_OF_DWORD
FUNCTION WORD_OF_DWORD : WORD
VAR_INPUT
	in : DWORD;
	N : BYTE;
END_VAR


(*
version 1.2	30. oct. 2008
programmer 	hugo
tested by	oscat

this function extracts a single word from the nth position from right (right is lowest byte)
the lower word (starting with Bit0 from in) is selected with N=0.
*)

WORD_OF_DWORD := DWORD_TO_WORD(SHR(in,SHL(n,4)));

(* revision history
hm	17. jan 2007	rev 1.0
	original version

hm	2. jan 2008		rev 1.1
	improved performance

hm	30. oct. 2008	rev 1.2
	improved performance
*)

END_FUNCTION

// oscat_basic/POUs/Logic/generators/A_TRIG
FUNCTION_BLOCK A_TRIG
VAR_INPUT
	IN : REAL;
	RES : REAL;
END_VAR
VAR_OUTPUT
	Q : BOOL;
	D : REAL;
END_VAR
VAR
	last_in : REAL;
END_VAR

(*
version 1.1	25. oct. 2008
programmer 	hugo
tested by	oscat

this block is similar to the IEC Standard R_trig and F_trig but it monitors a REAL for change.
if the valiue on IN changes more then D from the last value it will generate trigger and display the difference in output D.
the trigger will only be active for one cycle.

*)

D := IN - LAST_IN;
Q := ABS(D) > res;
IF Q THEN last_in := IN; END_IF;
D := IN - LAST_IN;


(* revision history

hm 	16. jul. 2008	rev 1.0
	original version released

hm	25. oct. 2008	rev 1.1
	code optimization
	a_trig now also works for res = 0

*)

END_FUNCTION_BLOCK

// oscat_basic/POUs/Logic/generators/B_TRIG
FUNCTION_BLOCK B_TRIG
VAR_INPUT
	CLK : BOOL;
END_VAR
VAR_OUTPUT
	Q : BOOL;
END_VAR
VAR
	edge : BOOL;
END_VAR

(*
version 1.0	4. aug. 2006
programmer 	hugo
tested by		tobias

this block is similar to R_trig and F_trig but it generates a pulse on rising and falling edge.

*)

Q := clk XOR edge;
edge := CLK;


(* revision history
hm		4. aug. 2006	rev 1.0
	original version

*)

END_FUNCTION_BLOCK

// oscat_basic/POUs/Logic/generators/CLICK_CNT
FUNCTION_BLOCK CLICK_CNT
VAR_INPUT
	IN : BOOL;
	N : INT;
	TC : TIME;
END_VAR
VAR_OUTPUT
	Q : BOOL;
END_VAR
VAR
	tx : TP;
	edge: BOOL;
	cnt: INT := -1;
END_VAR

(*
version 1.0	16. jul. 2008
programmer 	hugo
tested by	oscat

this Module decodes a specified number of clicks.
the output trig is high for one cycle if N clicks are present within a specified time TC.

*)

(* Q shall only be active for one cycle only *)
Q := FALSE;

IF in AND NOT edge AND NOT tx.q THEN
	(* a rising edge on in sets the counter to 0 *)
	cnt := 0;
ELSIF tx.Q AND NOT IN AND edge THEN
	(* count falling edges when tp.q is true *)
	cnt := cnt + 1;
ELSIF NOT tx.Q THEN
	Q := cnt = N;
	cnt := -1;
END_IF;

(* remember the status of IN *)
edge := IN;
tx(in := IN, pt := TC);


(* revision history

hm 	16. jul. 2008	rev 1.0
	original version released


*)

END_FUNCTION_BLOCK

// oscat_basic/POUs/Logic/generators/CLICK_DEC
FUNCTION_BLOCK CLICK_DEC
VAR_INPUT
	IN : BOOL;
	TC : TIME;
END_VAR
VAR_OUTPUT
	Q0, Q1, Q2, Q3 : BOOL;
END_VAR
VAR
	tx : TP;
	edge: BOOL;
	cnt: INT := -1;
END_VAR

(*
version 1.1	14. mar. 2009
programmer 	hugo
tested by		oscat

this Module detects a rising edge on In and decodes the amount of falling edges (Pulses) within a specified time TC.
the outputs Q0..Q3 will go true for one cycle and the amount of clicks within a specified time TC.
if only a rising egde is detected within TC Q0 will respond, Q1 for 1 pulse and so on..

*)

(* Q shall only be active for one cycle only *)
IF in = FALSE THEN
	Q0 := FALSE;
	Q1 := FALSE;
	Q2:= FALSE;
	Q3 := FALSE;
END_IF;

IF in AND NOT edge AND NOT tx.q THEN
	(* a rising edge on in sets the counter to 0 *)
	cnt := 0;
ELSIF tx.Q AND NOT IN AND edge THEN
	(* count falling edges when tp.q is true *)
	cnt := cnt + 1;
ELSIF NOT tx.Q THEN
	CASE cnt OF
		0 : Q0 := TRUE;
		1 : Q1 := TRUE;
		2 : Q2 := TRUE;
		3 : Q3 := TRUE;
	END_CASE;
	cnt := -1;
END_IF;

(* remember the status of IN *)
edge := IN;
tx(in := IN, pt := TC);



(* revision history

hm 17. jul. 2008	rev 1.0
	original version released

hm	14. mar. 2009	rev 1.1
	removed double assignments

*)

END_FUNCTION_BLOCK

// oscat_basic/POUs/Logic/generators/CLK_DIV
FUNCTION_BLOCK CLK_DIV
VAR_INPUT
	clk : BOOL;
	rst: BOOL;
END_VAR
VAR_OUTPUT
	Q0 : BOOL;
	Q1 : BOOL;
	Q2 : BOOL;
	Q3 : BOOL;
	Q4 : BOOL;
	Q5 : BOOL;
	Q6 : BOOL;
	Q7 : BOOL;
END_VAR
VAR
	cnt: BYTE;
END_VAR

(*
version 1.1	2 jan 2008
programmer 	hugo
tested by		tobias

this is a clock divider
each output divides the signal by 2
Q0 = clk / 2 , Q1 = Q0 / 2 and so on.
the outputs have a 50% duty cycle each.


*)

IF rst THEN
	cnt:= 0;
	Q0 := 0;
	Q1 := 0;
	Q2 := 0;
	Q3 := 0;
	Q4 := 0;
	Q5 := 0;
	Q6 := 0;
	Q7 := 0;
ELSIF clk THEN
	cnt:= cnt +1;
	Q0 := cnt.0;
	Q1 := cnt.1;
	Q2 := cnt.2;
	Q3 := cnt.3;
	Q4 := cnt.4;
	Q5 := cnt.5;
	Q6 := cnt.6;
	Q7 := cnt.7;
END_IF;

(* revision history
hm	4. aug. 2006	rev 1.0
	original version

hm	2. jan 2008		rev 1.1
	improved performance

*)

END_FUNCTION_BLOCK

// oscat_basic/POUs/Logic/generators/CLK_N
FUNCTION_BLOCK CLK_N
VAR_INPUT
	N : INT;
END_VAR
VAR_OUTPUT
	Q : BOOL;
END_VAR
VAR
	edge : BOOL;
	stime: DWORD;
	clk: BOOL;
END_VAR

(*
version 1.0	17 sep 2007
programmer 	hugo
tested by		tobias

clk_N uses the internal sps time to generate one pulse every N ms
every pulse is only valid for one cycle so that a edge trigger is not necessary
clk_N generates pulses depending on the accuracy of the system clock.
The input N controlls the period time of the clock.
N=0 equals 1ms, N=1 equals 2ms, N=2 equals 4ms, N=3 equals 8ms ....

be careful, 1ms clocks will only work on very powerful sps cpu's
*)

stime := SHR(T_PLC_MS(),N);
clk := stime.0;
Q := clk XOR edge;
edge := CLK;

(* revision history
hm	16. dec 2007		rev 1.0
	original version

*)

END_FUNCTION_BLOCK

// oscat_basic/POUs/Logic/generators/CLK_PULSE
FUNCTION_BLOCK CLK_PULSE
VAR_INPUT
	PT : TIME;
	N : INT;
	RST : BOOL ;
END_VAR
VAR_OUTPUT
	Q : BOOL;
	CNT : INT;
	RUN : BOOL;
END_VAR
VAR
	tx, tn: DWORD;
	init: BOOL;
END_VAR

(*
version 1.2		16 feb 2011
programmer 	hugo
tested by		oscat

clk_pulse uses the internal sps time to generate a clock with programmable period time.
the period time is defined for 10ms .. 65s.
pulse generation is continuous if N = 0 and for n pulses otherwise.
the first cycle after start is a clk pulse and then depending on the programmed period time a delay.
every pulse is only valid for one cycle so that a edge trigger is not necessary
clk_prg depending on the accuracy of the system clock.

*)

tx := T_PLC_MS();		(* read system *)
Q := FALSE;				(* reset Q we generate pulses only for one cycle *)
RUN := CNT < N;

IF NOT init OR RST THEN
	init := TRUE;
	CNT := 0;
	tn := tx - TIME_TO_DWORD(PT);
	RUN := FALSE;
ELSIF (cnt < N OR N = 0) AND tx - tn >= TIME_TO_DWORD(PT) THEN		(* generate a pulse *)
	CNT := CNT + 1;
	Q := TRUE;
	tn := tn + TIME_TO_DWORD(PT);
END_IF;



(* revision history
hm		4. aug 2006		rev 1.0
	original version

hm		17. sep 2007	rev 1.1
	replaced time() with T_PLC_S() for compatblity reasons

hm		16. feb. 2011	rev 1.2
	fixed an error when timer overflows 
*)

END_FUNCTION_BLOCK

// oscat_basic/POUs/Logic/generators/CYCLE_4
FUNCTION_BLOCK CYCLE_4
VAR_INPUT
	E : BOOL := TRUE;
	T0, T1, T2, T3 : TIME;
	S0 : BOOL;
	SX : INT;
	SL : BOOL;
END_VAR
VAR_OUTPUT
	STATE : INT;
END_VAR
VAR
	tx : TIME;
	last : TIME;
	init: BOOL;
END_VAR


(*
version 1.0	
programmer 	hugo
tested by	oscat


 
*)

(* read system timer *)
tx := DWORD_TO_TIME(T_PLC_MS());
(* init on first cycle *)
IF NOT init THEN
	init := TRUE;
	last := tx;
END_IF;

IF E THEN
	IF SL THEN
		(* when sx > 0 then the state sx is forced to start *)
		state:= LIMIT(0,SX,3);
		last := tx;
		(* this is to avoid to reset sx from the calling programm it does work fine on codesys but i am not sure about other systems, because we are writing to an input *)
		SL := FALSE;
	ELSE
		CASE state OF
			0 :	(* wait for T0 and switch to next cycle *)
				IF tx - last >= T0 THEN
					state := 1;
					last := tx;
				END_IF;
			1 : (* wait for T1 over 1st cycle *)
				IF tx - last >= T1 THEN
					state := 2;
					last := tx;
				END_IF;
			2 : (* wait for T1 over 1st cycle *)
				IF tx - last >= T2 THEN
					state := 3;
					last := tx;
				END_IF;
			3 : (* wait for T2 over 2nd cycle *)
				IF tx - last >= T3 THEN
					IF S0 THEN State := 0; END_IF; (* if S0 is false, the sequence stops at state 3 *)
					last := tx;
				END_IF;
		END_CASE;
	END_IF;
ELSE
	state := 0;
	last := tx;
END_IF;



(*
hm	3. nov. 2008	rev 1.0
	original version

*)

END_FUNCTION_BLOCK

// oscat_basic/POUs/Logic/generators/D_TRIG
FUNCTION_BLOCK D_TRIG
VAR_INPUT
	in : DWORD;
END_VAR
VAR_OUTPUT
	Q : BOOL;
	X : DWORD;
END_VAR
VAR
	last_in : DWORD;
END_VAR

(*
version 1.1	19. feb 2008
programmer 	hugo
tested by		tobias

this block is similar to the IEC Standard R_trig and F_trig but it monitors a DWORD, WORD or Byte Variable instead and generated an Output Pulse for one cycle only when the input has changed.
an additional output x (Dword) will state the chage of the input.
Example: the input has chaged from 0001 to 0010 then the output x will be 2.

*)

Q := in <> last_in;
X := in - last_in;
last_in := in;


(* revision history

hm 	4.09.2007		rev 1.0
	original version released

hm	19. feb. 2008	rev 1.1
	performance improvement
*)

END_FUNCTION_BLOCK

// oscat_basic/POUs/Logic/generators/GEN_BIT
FUNCTION_BLOCK GEN_BIT
VAR_INPUT
	in0 : DWORD;
	in1 : DWORD;
	in2 : DWORD;
	in3 : DWORD;
	clk : BOOL;
	steps : INT;
	rep : INT;
	rst : BOOL;
END_VAR
VAR_OUTPUT
	Q0 :BOOL;
	Q1 :BOOL;
	Q2 :BOOL;
	Q3 :BOOL;
	cnt : INT;
	run : BOOL;
END_VAR
VAR
	r0: DWORD;
	r1: DWORD;
	r2: DWORD;
	r3: DWORD;
	rx : INT := 1;
END_VAR

(*
version 1.2	14. mar. 2009
programmer 	hugo
tested by		tobias

gen_bit is 4 bit sequencial pattern generator with 4 DWORD inputs and 4 serial outputs.
with the first clock pulse after a reset or after power on, bit 0 of the input DWORDS IN is present on the Outputs Q and the next clock cycle shifts to Bit 1 and so on.
the input steps defines how many bits of the input dwords will be shifted to the outputs. the sequence can be repetive when rep = 0 or any amount of repetitions can be defined with input rep.

*)

(* check if number of runs is finished or rep = 0 which means continuous *)

IF clk AND NOT rst THEN
	run := (rep = 0) OR (rx <= rep);
	IF run THEN
		(* check for step counter reached and reset to 0 if cnt = steps *)
		IF cnt = steps THEN
			cnt := 0;
		END_IF;

		(* when cnt = 0 then reload the inputs into the registers *)
		IF cnt = 0 THEN
			r0 := in0;
			r1 := in1;
			r2 := in2;
			r3 := in3;
		END_IF;

		(* when cnt < steps, shift the lowest bits to the outputs *)
		IF (cnt < steps) THEN
			Q0 := r0.0;
			Q1 := r1.0;
			Q2 := r2.0;
			Q3 := r3.0;
			r0 := SHR(r0,1);
			r1 := SHR(r1,1);
			r2 := SHR(r2,1);
			r3 := SHR(r3,1);
		END_IF;

		(* increment the step counter *)
		cnt := cnt +1;
		IF (cnt = steps) AND (rep <> 0) THEN rx := rx +1; END_IF;
		IF (rx > rep) AND (rep <> 0) THEN run := FALSE; END_IF;
	END_IF;
ELSE
	IF rst THEN
		run := FALSE;
		Q0 := FALSE;
		Q1 := FALSE;
		Q2 := FALSE;
		Q3 := FALSE;
		r0 := 0;
		r1 := 0;
		r2 := 0;
		r3 := 0;
		cnt := 0;
		rx := 1;
	END_IF;
END_IF;



(* revision histroy
hm	4 aug 2006	rev 1.0
	original version

hm 15. oct. 2008	rev 1.1
	improved performance

hm	14. mar. 2009	rev 1.2
	removed double assignments

*)

END_FUNCTION_BLOCK

// oscat_basic/POUs/Logic/generators/GEN_SQ
FUNCTION_BLOCK GEN_SQ
VAR_INPUT
	PT : TIME;
END_VAR
VAR_OUTPUT
	Q : BOOL;
END_VAR
VAR
	tn: DWORD;
	tx: DWORD;
	init : BOOL;
END_VAR

(*
version 1.3	16. feb. 2011
programmer 	hugo
tested by		tobias

gen_sq generates square wave signal with programmable period time.

*)

(* read system time *)
tx := T_PLC_MS();

IF NOT init THEN
	init := TRUE;
	tn := tx;
	Q := TRUE;
ELSIF tx - tn >= SHR(TIME_TO_DWORD(PT),1) THEN
	Q := NOT Q;
	tn := tn + SHR(TIME_TO_DWORD(pt),1);
END_IF;


(* revision history
hm	4. aug 2006	rev 1.0
	original version

hm	17. sep 2007	rev 1.1
	replaced time() with T_PLC_MS() for compatibility reasons

hm	18. jul. 2009	rev 1.2
	improved accuracy

hm	16. feb 2011	rev 1.3
	corrected an error with timer overflow 
*)

END_FUNCTION_BLOCK

// oscat_basic/POUs/Logic/generators/SCHEDULER
FUNCTION_BLOCK SCHEDULER
VAR_INPUT
	E0 : BOOL;
	E1 : BOOL;
	E2 : BOOL;
	E3 : BOOL;
END_VAR
VAR_INPUT CONSTANT
	T0, T1, T2, T3 : TIME;
END_VAR
VAR_OUTPUT
	Q0, Q1, Q2, Q3 : BOOL;
END_VAR
VAR
	init : BOOL;
	s0, s1, s2, s3 : TIME;
	tx : TIME;
	c : INT;
END_VAR


(*
version 1.1	14. mar. 2009
programmer 	hugo
tested by		tobias

SCHEDULER is used to call programs or function blocks at specific intervals.
T0..T3 defines the interval times.

*)

(* read system_time *)
tx := DWORD_TO_TIME(T_PLC_MS());

IF NOT init THEN
	init := TRUE;
	s0 := tx - T0;
	s1 := tx - T1;
	s2 := tx - T2;
	s3 := tx - T3;
END_IF;

Q0 := FALSE;
Q1 := FALSE;
Q2 := FALSE;
Q3 :=FALSE;

CASE c OF
	0: 	IF tx - s0 >= T0 THEN
			Q0 := E0;
			s0 := tx;
		END_IF;
		c := 1;
	1: 	IF tx - s1 >= T1 THEN
			Q1 := E1;
			s1 := tx;
		END_IF;
		c := 2;
	2: 	IF tx - s2 >= T2 THEN
			Q2 := E2;
			s2 := tx;
		END_IF;
		c := 3;
	3: 	IF tx - s3 >= T3 THEN
			Q3 := E3;
			s3 := tx;
		END_IF;
		c := 0;
END_CASE;


(* revision history

hm 28. sep. 2008	rev 1.0
	original version

hm	14. mar. 2009	rev 1.1
	removed double assignments

*)

END_FUNCTION_BLOCK

// oscat_basic/POUs/Logic/generators/SCHEDULER_2
FUNCTION_BLOCK SCHEDULER_2
VAR_INPUT
	E0 : BOOL;
	E1 : BOOL;
	E2 : BOOL;
	E3 : BOOL;
END_VAR
VAR_INPUT CONSTANT
	C0, C1, C2, C3 : UINT;
	O0, O1, O2, O3 : UINT;
END_VAR
VAR_OUTPUT
	Q0, Q1, Q2, Q3 : BOOL;
END_VAR
VAR
	sx : UINT;
END_VAR


(*
version 1.0	29. sep 2008
programmer 	hugo
tested by		tobias

SCHEDULER_2 is used to call programs or function blocks at specific cycles.
C0..C3 defines after how many cycles the output becomes active.
O0..O3 defines a cycle offset at startup.

*)

Q0 := E0 AND (sx MOD C0 - O0 = 0);
Q1 := E1 AND (sx MOD C1 - O1 = 0);
Q2 := E2 AND (sx MOD C2 - O2 = 0);
Q3 := E3 AND (sx MOD C3 - O3 = 0);

(* increment cycle counter every cycle *)
sx := sx + 1;


(* revision history
hm 29. sep. 2008		rev 1.0
	original version


*)

END_FUNCTION_BLOCK

// oscat_basic/POUs/Logic/generators/SEQUENCE_4
FUNCTION_BLOCK SEQUENCE_4
VAR_INPUT
	in0 : BOOL := TRUE;
	in1 : BOOL := TRUE;
	in2 : BOOL := TRUE;
	in3 : BOOL := TRUE;
	start : BOOL;
	rst : BOOL;
	wait0 : TIME;
	delay0 : TIME;
	wait1 : TIME;
	delay1 : TIME;
	wait2 : TIME;
	delay2 : TIME;
	wait3 : TIME;
	delay3 : TIME;
END_VAR
VAR_INPUT CONSTANT
	stop_on_error : BOOL;
END_VAR
VAR_OUTPUT
	Q0 : BOOL;
	Q1 : BOOL;
	Q2 : BOOL;
	Q3 : BOOL;
	QX : BOOL;
	run: BOOL;
	step : INT := -1;
	status : BYTE;
END_VAR
VAR
	last : TIME;
	edge : BOOL;
	tx: TIME;
	init: BOOL;
END_VAR

(*
version 1.5	13. mar. 2009
programmer 	oscat
tested by		hans

sequence_4 enables run when a low to high transition is present on start.
a low to high transition on start will restart the sequencer at any time while a rst will hold the sequencer in reset while true.
after run is enabled with a rising edge on start the sequencer waits for wait0 on in0 to enable q0 which stays on for delay0.
the next cycle starts with wait1, continues with delay 1 and so on...
if an edge is not detected during the wait period, the sequencer will then display the error number on the status output.
the status numbers 1..4 are errors in step 0..3.
after the last step that sets q3, the sequencer leaves q3 on for delay3 and then resets to the initial state.
a step output will indicate the current step of the sequencer and will also be present with a fault condition.
after the first output is turened on the sequencer switches from q0 to q1 and so on, at any time there is only one output enabled.
if an input signal is not detected during a wait period, the sequencer will display the error number ( 1 for in0, 2 for in1 .... ).
when an error is present and the config variable stop_on_error is set then the sequencer will stop. otherwise it will continue.
The status output will also display 110 for waiting and 111 for sequence running.
*)

(* read sps timer *)
tx := DWORD_TO_TIME(T_PLC_MS());

(* initialize on startup *)
IF NOT init THEN
	last := tx;
	init := TRUE;
	status := 110;
END_IF;

(* asynchronous reset *)
IF rst THEN
	step := -1;
	Q0 := 0;
	Q1 := 0;
	Q2 := 0;
	Q3 := 0;
	status := 110;
	run := 0;

(* edge on start input restarts the sequencer *)
ELSIF start AND NOT edge THEN
	step := 0;
	last := tx;
	status := 111;
	Q0 := 0;
	Q1 := 0;
	Q2 := 0;
	Q3 := 0;
	run := 1;
END_IF;
edge := start;

(* check if stop on status is necessary *)
IF status > 0 AND status < 100 AND stop_on_error THEN RETURN; END_IF;

(* sequence is running *)
IF run AND step = 0 THEN
	IF NOT q0 AND in0 AND tx - last <= wait0 THEN
		Q0 := TRUE;
		last := tx;
	ELSIF NOT q0 AND tx - last > wait0 THEN
		status := 1;
		run := FALSE;
	ELSIF q0 AND tx - last >= delay0 THEN
		step := 1;
		last := tx;
	END_IF;
END_IF;
IF run AND step = 1 THEN
	IF NOT q1 AND in1 AND tx - last <= wait1 THEN
		Q0 := FALSE;
		Q1 := TRUE;
		last := tx;
	ELSIF NOT q1 AND Tx - last > wait1 THEN
		status := 2;
		q0 := FALSE;
		run := FALSE;
	ELSIF q1 AND tx - last >= delay1 THEN
		step := 2;
		last := tx;
	END_IF;
END_IF;
IF run AND step = 2 THEN
	IF NOT q2 AND in2 AND tx - last <= wait2 THEN
		Q1 := FALSE;
		Q2 := TRUE;
		last := tx;
	ELSIF NOT q2 AND Tx - last > wait2 THEN
		status := 3;
		q1 := FALSE;
		run := FALSE;
	ELSIF q2 AND tx - last >= delay2 THEN
		step := 3;
		last := tx;
	END_IF;
END_IF;
IF run AND step = 3 THEN
	IF NOT q3 AND in3 AND tx - last <= wait3 THEN
		Q2 := FALSE;
		Q3 := TRUE;
		last := tx;
	ELSIF NOT q3 AND Tx - last > wait3 THEN
		status := 4;
		q2 := FALSE;
		run := FALSE;
	ELSIF q3 AND tx - last >= delay3 THEN
		step := -1;
		q3 := FALSE;
		run := FALSE;
		status := 110;
	END_IF;
END_IF;
QX := q0 OR q1 OR q2 OR q3;

(*
hm 1.10.06		rev 1.1
	corrected delay logic to be after event and not before
	added any output

hm 1.12.06		rev 1.2
	corrected failure in sequence logic.
	added init at startup to prevent from initial error after start.

hm 17.1.2007		rev 1.3
	changed output fault to status for better compatibility with other modules (ESR).
	added stop on error functionality and setup variable
	default for inputs in0..3 is true.
	renamed variable state to step

hm	17.sep 2007	rev 1.4
	replaced time() with T_PLC_MS() for compatibility reasons

hm	13. mar. 2009	rev 1.5
	renamed output any to qx for compatibility resons

*)

END_FUNCTION_BLOCK

// oscat_basic/POUs/Logic/generators/SEQUENCE_64
FUNCTION_BLOCK SEQUENCE_64
VAR_INPUT
	START : BOOL;
	SMAX : INT;
	PROG : ARRAY[0..63]OF TIME;
	RST : BOOL;
END_VAR
VAR_OUTPUT
	STATE : INT := -1;
	TRIG : BOOL;
END_VAR
VAR
	tx : TIME;
	edge: BOOL;
	last: TIME;
END_VAR


(*
version 1.0	29. jun. 2008
programmer 	hugo
tested by	oscat

sequence generates a sequence of states with a programmable length for each state.

*)

(* read system timer *)
tx := DWORD_TO_TIME(T_PLC_MS());
TRIG := FALSE;

IF RST THEN
	STATE := -1;

(* start sequence *)
ELSIF START AND NOT edge THEN
	STATE := 0;
	last := tx;
	TRIG := TRUE;

(* sequence generator *)
ELSIF (STATE >= 0) THEN
	IF (tx - last) >= PROG[STATE] THEN
		STATE := INC2(STATE, 1, -1, SMAX);
		last := tx;
		TRIG := TRUE;
	END_IF;
END_IF;

edge := START;



(* revision history
hm	29. jun. 2008
	original version

*)

END_FUNCTION_BLOCK

// oscat_basic/POUs/Mathematical/INC2
FUNCTION INC2 : INT
VAR_INPUT
	X : INT;
	D : INT;
	L : INT;
	U : INT;
END_VAR
VAR
	tmp: INT;
END_VAR


(*
version 1.0	29. jun. 2008
programmer 	hugo
tested by	oscat

This function increments the input X by the value D and compares the result with U.
if the output exceeds U it will continue to count from L again.

*)

tmp := U - L + 1;
INC2 := (X + D - L + tmp) MOD tmp + L;



(* revision history
hm	29. jun. 2008		REV 1.0
	original version


*)

END_FUNCTION

// oscat_basic/POUs/Logic/generators/SEQUENCE_8
FUNCTION_BLOCK SEQUENCE_8
VAR_INPUT
	in0 : BOOL := TRUE;
	in1 : BOOL := TRUE;
	in2 : BOOL := TRUE;
	in3 : BOOL := TRUE;
	in4 : BOOL := TRUE;
	in5 : BOOL := TRUE;
	in6 : BOOL := TRUE;
	in7 : BOOL := TRUE;
	start : BOOL;
	rst : BOOL;
	wait0 : TIME;
	delay0 : TIME;
	wait1 : TIME;
	delay1 : TIME;
	wait2 : TIME;
	delay2 : TIME;
	wait3 : TIME;
	delay3 : TIME;
	wait4 : TIME;
	delay4 : TIME;
	wait5 : TIME;
	delay5 : TIME;
	wait6 : TIME;
	delay6 : TIME;
	wait7 : TIME;
	delay7 : TIME;
END_VAR
VAR_INPUT CONSTANT
	stop_on_error : BOOL;
END_VAR
VAR_OUTPUT
	Q0 : BOOL;
	Q1 : BOOL;
	Q2 : BOOL;
	Q3 : BOOL;
	Q4 : BOOL;
	Q5 : BOOL;
	Q6 : BOOL;
	Q7 : BOOL;
	QX : BOOL;
	run: BOOL;
	step : INT := -1;
	status : BYTE;
END_VAR
VAR
	last : TIME;
	edge : BOOL;
	tx: TIME;
	init: BOOL;
END_VAR

(*
version 1.5	13. mar. 2009
programmer 	oscat
tested by		hans

sequence_8 enables run when a low to high transition is present on start.
a low to high transition on start will restart the sequencer at any time while a rst will hold the sequencer in reset while true.
after run is enabled with a rising edge on start the sequencer waits for wait0 on in0 to enable q0 which stays on for delay0.
the next cycle starts with wait1, continues with delay 1 and so on...
if an edge is not detected during the wait period, the sequencer will then display the error number on the status output.
The status numbers are 1 .. 8 for erros in step 0..7.
after the last step that sets q7, the sequencer leaves q7 on for delay7 and then resets to the initial state.
a step output will indicate the current step of the sequencer and will also be present with a fault condition.
after the first output is turened on the sequencer switches from q0 to q1 and so on, at any time there is only one output enabled.
if an input signal is not detected during a wait period, the sequencer will display the error number ( 1 for in0, 2 for in1 .... ).
when an error is present and the config variable stop_on_error is set then the sequencer will stop. otherwise it will continue.
The status output will also display 110 for waiting and 111 sequece running.

*)

(* read sps timer *)
tx := DWORD_TO_TIME(T_PLC_MS());

(* initialize on startup *)
IF NOT init THEN
	last := tx;
	init := TRUE;
	status := 110;
END_IF;

(* asynchronous reset *)
IF rst THEN
	step := -1;
	Q0 := 0;
	Q1 := 0;
	Q2 := 0;
	Q3 := 0;
	Q4 := 0;
	Q5 := 0;
	Q6 := 0;
	Q7 := 0;
	status := 110;
	run := 0;

(* edge on start input restarts the sequencer *)
ELSIF start AND NOT edge THEN
	step := 0;
	last := tx;
	status := 111;
	Q0 := 0;
	Q1 := 0;
	Q2 := 0;
	Q3 := 0;
	Q4 := 0;
	Q5 := 0;
	Q6 := 0;
	Q7 := 0;
	run := 1;
END_IF;
edge := start;

(* check if stop on error is necessary *)
IF status > 0 AND status < 100 AND stop_on_error THEN RETURN; END_IF;

(* sequence is running *)
IF run AND step = 0 THEN
	IF NOT q0 AND in0 AND tx - last <= wait0 THEN
		Q0 := TRUE;
		last := tx;
	ELSIF NOT q0 AND tx - last > wait0 THEN
		status := 1;
		run := FALSE;
	ELSIF q0 AND tx - last >= delay0 THEN
		step := 1;
		last := tx;
	END_IF;
END_IF;
IF run AND step = 1 THEN
	IF NOT q1 AND in1 AND tx - last <= wait1 THEN
		Q0 := FALSE;
		Q1 := TRUE;
		last := tx;
	ELSIF NOT q1 AND Tx - last > wait1 THEN
		status := 2;
		q0 := FALSE;
		run := FALSE;
	ELSIF q1 AND tx - last >= delay1 THEN
		step := 2;
		last := tx;
	END_IF;
END_IF;
IF run AND step = 2 THEN
	IF NOT q2 AND in2 AND tx - last <= wait2 THEN
		Q1 := FALSE;
		Q2 := TRUE;
		last := tx;
	ELSIF NOT q2 AND Tx - last > wait2 THEN
		status := 3;
		q1 := FALSE;
		run := FALSE;
	ELSIF q2 AND tx - last >= delay2 THEN
		step := 3;
		last := tx;
	END_IF;
END_IF;
IF run AND step = 3 THEN
	IF NOT q3 AND in3 AND tx - last <= wait3 THEN
		Q2 := FALSE;
		Q3 := TRUE;
		last := tx;
	ELSIF NOT q3 AND Tx - last > wait3 THEN
		status := 4;
		q2 := FALSE;
		run := FALSE;
	ELSIF q3 AND tx - last >= delay3 THEN
		step := 4;
		last := tx;
	END_IF;
END_IF;
IF run AND step = 4 THEN
	IF NOT q4 AND in4 AND tx - last <= wait4 THEN
		Q3 := FALSE;
		Q4 := TRUE;
		last := tx;
	ELSIF NOT q4 AND Tx - last > wait4 THEN
		status := 5;
		q3 := FALSE;
		run := FALSE;
	ELSIF q4 AND tx - last >= delay4 THEN
		step := 5;
		last := tx;
	END_IF;
END_IF;
IF run AND step = 5 THEN
	IF NOT q5 AND in5 AND tx - last <= wait5 THEN
		Q4 := FALSE;
		Q5 := TRUE;
		last := tx;
	ELSIF NOT q5 AND Tx - last > wait5 THEN
		status := 6;
		q4 := FALSE;
		run := FALSE;
	ELSIF q5 AND tx - last >= delay5 THEN
		step := 6;
		last := tx;
	END_IF;
END_IF;
IF run AND step = 6 THEN
	IF NOT q6 AND in6 AND tx - last <= wait6 THEN
		Q5 := FALSE;
		Q6 := TRUE;
		last := tx;
	ELSIF NOT q6 AND Tx - last > wait6 THEN
		status := 7;
		q5 := FALSE;
		run := FALSE;
	ELSIF q6 AND tx - last >= delay6 THEN
		step := 7;
		last := tx;
	END_IF;
END_IF;
IF run AND step = 7 THEN
	IF NOT q7 AND in7 AND tx - last <= wait7 THEN
		Q6 := FALSE;
		Q7 := TRUE;
		last := tx;
	ELSIF NOT q7 AND Tx - last > wait7 THEN
		status := 8;
		q6 := FALSE;
		run := FALSE;
	ELSIF q7 AND tx - last >= delay7 THEN
		step := -1;
		Q7 := FALSE;
		Run := FALSE;
		status := 110;
	END_IF;
END_IF;
QX := q0 OR q1 OR q2 OR q3 OR q4 OR q5 OR q6 OR q7;

(*
hm 1.10.06		rev 1.1
	corrected delay logic to be after event and not before
	added any output

hm 1.12.06		rev 1.2
	corrected failure in sequence logic.
	added init at startup to prevent from initial statuss after start.

hm 17.1.2007		rev 1.3
	changed output fault to status for better compatibility with other modules (ESR)
	added stop on error functionality and setup variable
	default for inputs in0..7 is true.
	renames variable state to step

hm	17.sep 2007	rev 1.4
	replaced time() with T_PLC_MS() for compatibility reasons

hm	13. mar. 2009	rev 1.5
	renamed output any to qx for compatibility resons

*)

END_FUNCTION_BLOCK

// oscat_basic/POUs/Logic/generators/TMIN
FUNCTION_BLOCK TMIN
VAR_INPUT
	IN : BOOL;
	PT : TIME;
END_VAR
VAR_OUTPUT
	Q : BOOL;
END_VAR
VAR
	pm : TP;
END_VAR

(*
version 1.0	21. jul. 2008
programmer 	hugo
tested by	oscat

Q of tMIN will follow IN except that it forces a minimum ontime for the output Q.

*)

pm(in := IN, PT := PT);
Q := IN OR pm.Q;


(* revision history
hm	21. jul. 2008	rev 1.0
	original version

*)

END_FUNCTION_BLOCK

// oscat_basic/POUs/Logic/generators/TOF_1
FUNCTION_BLOCK TOF_1
VAR_INPUT
	IN : BOOL;
	PT : TIME;
	RST : BOOL;
END_VAR
VAR_OUTPUT
	Q : BOOL;
END_VAR
VAR
	tx : TIME;
	start : TIME;
END_VAR

(*
version 1.0	17. jul. 2008
programmer 	hugo
tested by	oscat

TOF_1 will extend a pulse on input in for PT seconds.
in addition the timer can be cleared asynchronously with rst.
TOF_1 is the same function as TOF from the standard LIB except the asynchronous reset input.

*)

(* read system timer *)
tx := DWORD_TO_TIME(T_PLC_MS());

IF RST THEN
	Q := FALSE;
ELSIF IN THEN
	Q := TRUE;
	start := tx;
ELSIF tx - start >= PT THEN
	Q := FALSE;
END_IF;




(* revision history
hm	17. jul. 2008	rev 1.0
	original version

*)

END_FUNCTION_BLOCK

// oscat_basic/POUs/Logic/generators/TONOF
FUNCTION_BLOCK TONOF
VAR_INPUT
	IN : BOOL;
	  T_ON,T_OFF : TIME;
END_VAR
VAR_OUTPUT
	Q : BOOL;
END_VAR
VAR
   X : TON;
   old: BOOL;
   mode: BOOL;
END_VAR

(*
version 1.2	21. jul 2009
programmer 	hugo
tested by		tobias

TONOF generated a TON and TOF Delay for the Input N TON (T1) and TOF (T2) can be configured separately
*)

IF IN XOR old THEN
  X(IN := FALSE, PT := SEL(IN,T_OFF,T_ON));
  mode := IN;
  old := IN;
END_IF;
X(IN := TRUE);
IF X.Q THEN Q := mode;END_IF;

(* revision history
hm	10. dec 2007	rev 1.0
	original version

hm	17. sep. 2007	rev 1.1
	improved performance

hm	21. jul. 2009	rev 1.2
	fixed a timing probelm


*)

END_FUNCTION_BLOCK

// oscat_basic/POUs/Logic/generators/TP_1
FUNCTION_BLOCK TP_1
VAR_INPUT
	IN : BOOL;
	PT : TIME;
	RST : BOOL;
END_VAR
VAR_OUTPUT
	Q : BOOL;
END_VAR
VAR
	tx : TIME;
	start : TIME;
	ix : BOOL;
END_VAR

(*
version 1.0	28. jun. 2008
programmer 	hugo
tested by		oscat

TP_1 generates a pulse every time it is calles with in := TRUE.
in addition the timer can be cleared asynchronously with rst.
the timer can be retriggered as often as necessary. it will count PT from the last trigger.

*)

(* read system timer *)
tx := DWORD_TO_TIME(T_PLC_MS());

IF RST THEN
	Q := FALSE;
ELSIF IN AND NOT ix THEN
	Q := TRUE;
	start := tx;
ELSIF tx - start >= PT THEN
	Q := FALSE;
END_IF;

ix:= IN;



(* revision history
hm	28. jun. 2008
	original version

*)

END_FUNCTION_BLOCK

// oscat_basic/POUs/Logic/memory/FIFO_16
FUNCTION_BLOCK FIFO_16
VAR_INPUT
	Din : DWORD;
	E : BOOL := TRUE;
	RD : BOOL;
	WD : BOOL;
	RST : BOOL;
END_VAR
VAR_OUTPUT
	Dout : DWORD;
	EMPTY : BOOL := TRUE;
	FULL : BOOL;
END_VAR
VAR
	fifo : ARRAY[0..n] OF DWORD;
	pr : INT;
	pw : INT;
END_VAR
VAR CONSTANT
	n : INT := 16;	(* changing this value will chage the number of stored elements in the fifo *)
END_VAR


(*
version 2.0	24. jul. 2009
programmer 	hugo
tested by		oscat

16 Dword FIFO memory
*)

IF RST THEN
	pw := pr;
	FULL := FALSE;
	EMPTY := TRUE;
	Dout := 0;
ELSIF E THEN
	IF NOT EMPTY AND RD THEN
		Dout := fifo[pr];
		pr := INC1(pr,n);
		EMPTY := pr = pw;
		FULL := FALSE;
	END_IF;
	IF NOT FULL AND WD THEN
		fifo[pw] := Din;
		pw := INC1(pw,n);
		FULL := pw = pr;
		EMPTY := FALSE;
	END_IF;
END_IF;


(* revision history

hm	4. aug. 2006	rev 1.0
	original version

hm	19. feb 2008	rev 1.1
	performance improvements

hm	17. oct. 2008	rev 1.2
	improved performance

ks	27. oct. 2008	rev 1.3
	optimized coding

hm	14. mar. 2009	rev 1.4
	removed double assignments

hm 24. jul. 2009	rev 2.0
	chaged inputs E and WR to E, WD and WR
	allow read and write in one cycle

*)

END_FUNCTION_BLOCK

// oscat_basic/POUs/Logic/memory/FIFO_32
FUNCTION_BLOCK FIFO_32
VAR_INPUT
	Din : DWORD;
	E : BOOL := TRUE;
	RD : BOOL;
	WD : BOOL;
	RST : BOOL;
END_VAR
VAR_OUTPUT
	Dout : DWORD;
	EMPTY : BOOL := TRUE;
	FULL : BOOL;
END_VAR
VAR
	fifo : ARRAY[0..n] OF DWORD;
	pr : INT;
	pw : INT;
END_VAR
VAR CONSTANT
	n : INT := 32;	(* changing this value will chage the number of stored elements in the fifo *)
END_VAR

(*
version 2.0	24. jul. 2009
programmer 	hugo
tested by		oscat

32 Dword FIFO memory
*)

IF RST THEN
	pw := pr;
	FULL := FALSE;
	EMPTY := TRUE;
	Dout := 0;
ELSIF E THEN
	IF NOT EMPTY AND RD THEN
		Dout := fifo[pr];
		pr := INC1(pr,n);
		EMPTY := pr = pw;
		FULL := FALSE;
	END_IF;
	IF NOT FULL AND WD THEN
		fifo[pw] := Din;
		pw := INC1(pw,n);
		FULL := pw = pr;
		EMPTY := FALSE;
	END_IF;
END_IF;

(* revision history
hm	4. aug. 2006	rev 1.0
	original version

hm	19. feb 2008	rev 1.1
	performance improvements

hm	17. oct. 2008	rev 1.2
	improved performance

ks	27. oct. 2008 rev 1.3
	improved code

hm	14. mar. 2009	rev 1.4
	removed double assignments

hm 24. jul. 2009	rev 2.0
	chaged inputs E and WR to E, WD and WR
	allow read and write in one cycle

*)

END_FUNCTION_BLOCK

// oscat_basic/POUs/Logic/memory/STACK_16
FUNCTION_BLOCK STACK_16
VAR_INPUT
	Din : DWORD;
	E : BOOL := TRUE;
	RD : BOOL;
	WD : BOOL;
	RST : BOOL;
END_VAR
VAR_OUTPUT
	Dout : DWORD;
	EMPTY : BOOL := TRUE;
	FULL : BOOL;
END_VAR
VAR
	stack : ARRAY[0..n] OF DWORD;
	pt : INT;
END_VAR
VAR CONSTANT
	n : INT := 15;	(* changing this value will chage the number of stored elements in the fifo *)
END_VAR


(*
version 2.0	25. jul 2009
programmer 	hugo
tested by		oscat

16 Dword STACK memory

*)

IF RST THEN
	(* asynchronous reset for the fifo *)
	pt := 0;
	EMPTY := TRUE;
	FULL := FALSE;
	Dout := 0;
ELSIF E THEN
	IF NOT EMPTY AND RD THEN
		(* read one element *)
		pt := pt - 1;
		Dout := stack[pt];
		EMPTY := pt = 0;
		FULL := FALSE;
	END_IF;
	IF NOT FULL AND WD THEN
		(* write one element *)
		stack[pt] := Din;
		pt := pt + 1;
		FULL := pt > n;
		EMPTY := FALSE;
	END_IF;
END_IF;


(* revision history
hm	4. aug. 2006	rev 1.0
	original version

hm	19. feb 2008	rev 1.1
	performance improvements

hm	17. oct. 2008	rev 1.2
	deleted unnecessary init with 0

hm	27. oct. 2008	rev 1.3
	optimized performance

hm	25. jul 2009	rev 2.0
	changed inputs to allow simultsaneous read and write
*)

END_FUNCTION_BLOCK

// oscat_basic/POUs/Logic/memory/STACK_32
FUNCTION_BLOCK STACK_32
VAR_INPUT
	Din : DWORD;
	E : BOOL := TRUE;
	RD : BOOL;
	WD : BOOL;
	RST : BOOL;
END_VAR
VAR_OUTPUT
	Dout : DWORD;
	EMPTY : BOOL := TRUE;
	FULL : BOOL;
END_VAR
VAR
	stack : ARRAY[0..n] OF DWORD;
	pt : INT;
END_VAR
VAR CONSTANT
	n : INT := 31;	(* changing this value will chage the number of stored elements in the fifo *)
END_VAR


(*
version 2.0	25. jul 2009
programmer 	hugo
tested by		oscat

32 Dword STACK memory
*)

IF RST THEN
	(* asynchronous reset for the fifo *)
	pt := 0;
	EMPTY := TRUE;
	FULL := FALSE;
	Dout := 0;
ELSIF E THEN
	IF NOT EMPTY AND RD THEN
		(* read one element *)
		pt := pt - 1;
		Dout := stack[pt];
		EMPTY := pt = 0;
		FULL := FALSE;
	END_IF;
	IF NOT FULL AND WD THEN
		(* write one element *)
		stack[pt] := Din;
		pt := pt + 1;
		FULL := pt > n;
		EMPTY := FALSE;
	END_IF;
END_IF;


(* revision history
hm	4. aug. 2006	rev 1.0
	original version

hm	19. feb 2008	rev 1.1
	performance improvements

hm	17. oct. 2008	rev 1.2
	deleted unnecessary init with 0

ks	27. oct. 2008	rev 1.3
	optimized performance

hm	25. jul 2009	rev 2.0
	changed inputs to allow simultsaneous read and write

*)

END_FUNCTION_BLOCK

// oscat_basic/POUs/Logic/Others/CRC_GEN
FUNCTION CRC_GEN : DWORD

VAR_INPUT
	PT : POINTER TO ARRAY[0..32000] OF BYTE;
	SIZE : INT;
	PL : INT;
	PN : DWORD;
	INIT : DWORD;
	REV_IN : BOOL;
	REV_OUT : BOOL;
	XOR_OUT : DWORD;
END_VAR
VAR
	pos : INT;
	shift : INT;
	dx: BYTE;
	bits: INT;
END_VAR

(*
version 2.0	16.Jan. 2011
programmer 	hugo
tested by		tobias

CRC_GEN generates a CRC checksum from a block of data and returns  the checksum in a DWORD to be connected to the data for transmission.
the CRC Polynom is specified with the config variable PN and the length of the Polynom is specified by PL
A Polynom x4 + X + 1 is represented by 0011 with length 4, the highest order bit is not specified at all..
The input data is an array of byte of any size, the function is called by CRC_GEN(ADR(array),SIZEOF(array), ....).

*)

(* align polygon *)
shift := 32 - PL;
PN := SHL(PN, shift);

(* load first 4 bytes into register minimum message size is 4 bytes
	for smaller messages fill with 0#s at the beginning*)
FOR pos := 0 TO 3 DO
	IF REV_IN THEN CRC_GEN := SHL(CRC_GEN, 8) OR REVERSE(PT^[pos]); ELSE CRC_GEN := SHL(CRC_GEN, 8) OR PT^[pos]; END_IF;
END_FOR;
pos := 4;

(* xor with init value *)
CRC_GEN := CRC_GEN XOR SHL(init, shift);

(* calculate CRC for each byte *)
WHILE pos < size DO
	IF REV_IN THEN DX := REVERSE(PT^[pos]); ELSE DX := PT^[pos]; END_IF;
	pos := pos + 1;
	(* crc calculation for one byte *)
	FOR bits := 0 TO 7 DO
		IF CRC_GEN.31 THEN
			CRC_GEN := (SHL(CRC_GEN, 1) OR BOOL_TO_DWORD(DX.7)) XOR PN;
		ELSE
			CRC_GEN := SHL(CRC_GEN, 1) OR BOOL_TO_DWORD(DX.7);
		END_IF;
		dx := SHL(dx, 1);
	END_FOR;
END_WHILE;

(* all bytes are processed, need to finish the registers 32 bits *)
FOR bits := 0 TO 31 DO
	IF CRC_GEN.31 THEN
		CRC_GEN := (SHL(CRC_GEN, 1) OR BOOL_TO_DWORD(DX.7)) XOR PN;
	ELSE
		CRC_GEN := SHL(CRC_GEN, 1) OR BOOL_TO_DWORD(DX.7);
	END_IF;
END_FOR;

(* final XOR *)
CRC_GEN := SHR(CRC_GEN, shift) XOR XOR_OUT;

(* reverse the crc_out put if necessary *)
IF REV_OUT THEN CRC_GEN := REFLECT(CRC_GEN, PL); END_IF;


(* typical crc polynoms

CRC-4-ITU 			x4 + x + 1 					(ITU G.704, p. 12) 	0x3 or 0xC (0x9)
CRC-5-ITU 			x5 + x4 + x2 + 1 			(ITU G.704, p. 9) 	0x15 or 0x15 (0x0B) Bluetooth
CRC-5-USB 			x5 + x2 + 1 				(use: USB token packets) 	0x05 or 0x14 (0x9)
CRC-6-ITU 			x6 + x + 1 					(ITU G.704, p. 3) 	0x03 or 0x30 (0x21)
CRC-7 				x7 + x3 + 1 				(use: telecom systems, MMC) 	0x09 or 0x48 (0x11)
CRC-8-ATM 			x8 + x2 + x + 1 				(use: ATM HEC) 	0x07 or 0xE0 (0xC1)
CRC-8-CCITT 		x8 + x7 + x3 + x2 + 1 		(use: 1-Wire bus) 	0x8D or 0xB1 (0x63)
CRC-8-Dallas/Maxim 	x8 + x5 + x4 + 1 			(use: 1-Wire bus) 	0x31 or 0x8C (0x19)
CRC-8 				x8 + x7 + x6 + x4 + x2 + 1 	0xD5 or 0xAB (0x57)
CRC-8-SAE J1850 	x8 + x4 + x3 + x2 + 1 		0x1D or 0xB8
CRC-10 				x10 + x9 + x5 + x4 + x + 1 	0x233 or 0x331 (0x263)
CRC-12 				x12 + x11 + x3 + x2 + x + 1 (use: telecom systems) 	0x80F or 0xF01 (0xE03)
CRC-15-CAN 			x15 + x14 + x10 + x8 + x7 + x4 + x3 + 1 	0x4599 or 0x4CD1 (0x19A3)
CRC-16-Fletcher 	Not a CRC; see Fletcher's checksum 	Used in Adler-32 A & B CRCs
CRC-16-CCITT 	x16 + x12 + x5 + 1 (XMODEM,X.25, V.41, Bluetooth, PPP, IrDA; known as "CRC-CCITT") 	0x1021 or 0x8408 (0x0811)
CRC-16-IBM 	x16 + x15 + x2 + 1 (USB, many others; also known as "CRC-16") 	0x8005 or 0xA001 (0x4003)
CRC-24-Radix-64 	x24 + x23 + x18 + x17 + x14 + x11 + x10 + x7 + x6 + x5 + x4 + x3 + x + 1 	0x864CFB or 0xDF3261 (0xBE64C3)
CRC-32-Adler 	Not a CRC; see Adler-32 	See Adler-32
CRC-32-MPEG2 	x32 + x26 + x23 + x22 + x16 + x12 + x11 + x10 + x8 + x7 + x5 + x4 + x2 + x + 1 	0x04C11DB7 or 0xEDB88320 (0xDB710641) Also used in IEEE 802.3
CRC-32-IEEE 802.3 	x32 + x26 + x23 + x22 + x16 + x12 + x11 + x10 + x8 + x7 + x5 + x4 + x2 + x + 1 (V.42) 	0x04C11DB7 or 0xEDB88320 (0xDB710641)
CRC-32C (Castagnoli) 	x32 + x28 + x27 + x26 + x25 + x23 + x22 + x20 + x19 + x18 + x14 + x13 + x11 + x10 + x9 + x8 + x6 + 1 	0x1EDC6F41 or 0x82F63B78 (0x05EC76F1)
CRC-64-ISO 	x64 + x4 + x3 + x + 1 (use: ISO 3309) 	0x000000000000001B or 0xD800000000000000 (0xB000000000000001)
CRC-64-ECMA-182 	x64 + x62 + x57 + x55 + x54 + x53 + x52 + x47 + x46 + x45 + x40 + x39 + x38 + x37 + x35 + x33 + x32 + x31 + x29 + x27 + x24 + x23 + x22 + x21 + x19 + x17 + x13 + x12 + x10 + x9 + x7 + x4 + x + 1
(as described in ECMA-182 p.63) 	0x42F0E1EBA9EA3693 or 0xC96C5795D7870F42 (0x92D8AF2BAF0E1E85)
*)



(* revision history

hm	9.6.2007		rev 1.0		
	original version 

hm	11.9.2007		rev 1.1
	deleted unused variable i

hm	9. oct 2007 	rev 1.2
	added init code for crc and xor_out
	added refelct in and reflect_out (rev_in und Rev_out)

hm	2. jan 2008	rev 1.3
	small changes for performance improvements

hm	16. mar. 2008	rev 1.4
	changed type of input size to uint

hm	10. mar. 2009	rev 1.5
	removed nested comments

hm	16. jan. 2011	rev 2.0
	new version
*)

END_FUNCTION

// oscat_basic/POUs/String/FILL
FUNCTION FILL : STRING(STRING_LENGTH)
VAR_INPUT
	C : BYTE;
	L : INT;
END_VAR
VAR
	i: INT;
	sx: STRING(1);
END_VAR

(*
version 1.1	17. dec. 2008
programmer 	hugo
tested by		tobias

the function fill creates a string at length L of characters C.

*)

Sx := CHR_TO_STRING(c);
(* limit L to maximum 80 characters the length of a standard string *)
L := LIMIT(0,L,STRING_LENGTH);
(* create a string of characters to be connected to str *)
FOR i := 1 TO 8 DO
	FILL := CONCAT(FILL,FILL);
	IF L.7 THEN FILL := CONCAT(FILL,Sx); END_IF;
	L := SHL(L,1);
END_FOR;




(* revision histroy
hm	29. mar. 2008	rev 1.0
	original release

hm	17. dec. 2008	rev 1.1
	changed function chr to chr_to_string

*)

END_FUNCTION

// oscat_basic/POUs/Logic/Others/MATRIX
FUNCTION_BLOCK MATRIX
VAR_INPUT
	x1, x2, x3, x4, X5 : BOOL;
END_VAR
VAR_INPUT CONSTANT
	Release : BOOL;
END_VAR
VAR_OUTPUT
	code : BYTE;
	TP : BOOL;
	y1: BOOL := TRUE;
	y2, y3, y4 : BOOL;
END_VAR
VAR
	line : BYTE;
	X : ARRAY[0..3] OF BYTE; (* scan line inputs *)
	L : ARRAY[0..3] OF BYTE; (* scan line status *)
	i: INT;
	temp: BYTE;
END_VAR

(*
version 1.3	26 oct. 2008
programmer 	hugo
tested by	oscat

MATRIX is a matrix keyboard encoder for 4 rows and up to 5 columns.
matrix can send a code while a key is pressed and it sends another code while a key is released when the setup variable 'release' is set to true.
the setup variable release is false the code is only sent when the key is pressed.
the output byte holds the 5 columns in the lowest bits 0..2  and the row number in bits 4..6, while bit 7 is true for a key pressed and false for a key released.

*)

TP := FALSE;
CODE := 0;
(* read scan lines *)
X[line].0 := X1;
X[line].1 := X2;
X[line].2 := X3;
X[line].3 := X4;
X[line].4 := X5;

(* compare for change *)
FOR i := 0 TO 3 DO
	IF X[i] <> L[i] THEN
		(* scan line information has changed code need to be found and generated *)
		temp := x[i] XOR L[i];
		IF temp.0 THEN
			CODE := 1;
			code.7 := X[i].0;
			L[i].0 := X[i].0;
		ELSIF temp.1 THEN
			code := 2;
			code.7 := X[i].1;
			L[i].1 := X[i].1;
		ELSIF temp.2 THEN
			code := 3;
			code.7 := X[i].2;
			L[i].2 := X[i].2;
		ELSIF temp.3 THEN
			CODE := 4;
			CODE.7 := X[i].3;
			L[i].3 := X[i].3;
		ELSIF temp.4 THEN
			CODE := 5;
			CODE.7 := X[i].4;
			L[i].4 := X[i].4;
		END_IF;
		TP := TRUE;
		CODE.4 := Line.0;
		CODE.5 := Line.1;
		CODE.6 := Line.2;

		(* check if release codes need to be killed *)
		IF NOT release AND CODE < 127 THEN
			CODE := 0;
			TP := FALSE;
		END_IF;
		EXIT;
	END_IF;
END_FOR;

(* increment scan line every cycle *)
line := (line + 1) AND 2#0000_0011;
temp := SHL(BYTE#1,line);
Y1 := temp.0;
Y2 := temp.1;
Y3 := temp.2;
Y4 := temp.3;




(* revision history
hm		10.6.2007	rev 1.0		
	original version 


hm		11.9.2007	rev 1.1		
	deleted unused variables k and old_code

hm		23.12.2007	rev 1.2
	added exit statement in for loop instead of i:=5

hm		26. oct. 2008	rev 1.3
	code optimized

*)

END_FUNCTION_BLOCK

// oscat_basic/POUs/Logic/Others/PIN_CODE
FUNCTION_BLOCK PIN_CODE
VAR_INPUT
	CB : BYTE;
	E : BOOL;
END_VAR
VAR_INPUT CONSTANT
	PIN : STRING(8);
END_VAR
VAR_OUTPUT
	TP : BOOL;
END_VAR
VAR
	POS: INT := 1;
END_VAR

(*
version 1.0	30. oct. 2008
programmer 	hugo
tested by	oscat

MATRIX_CODE scans the input of a key_pad (MATRIX) for a sequence of characters.

*)

tp := FALSE;
IF e THEN
	IF CB = CODE(pin, pos) THEN
		pos := pos + 1;
		IF pos > LEN(PIN) THEN
			(* proper code is detected *)
			TP := TRUE;
			pos := 1;
		END_IF;
	ELSE
		pos := 1;
	END_IF;
END_IF;


(* revision history
hm	30. oct. 2008	rev 1.0		
	original version 


*)

END_FUNCTION_BLOCK

// oscat_basic/POUs/Mathematical/Array/_ARRAY_ABS
FUNCTION _ARRAY_ABS : BOOL
VAR_INPUT
	pt : POINTER TO ARRAY[0..32000] OF REAL;
	size : UINT;
END_VAR
VAR
	i: UINT;
	stop: UINT;
END_VAR

(*
version 1.0	2. apr. 2008
programmer 	hugo
tested by	tobias

this function will calculate the absolute value of each element of the array and stroe the result instead of the element.
Array[i] := ABS(ARRAY[i]).
the function needs to be called:	array_avg(adr("array"),sizeof("array"));
because this function works with pointers its very time efficient and it needs no extra memory.

*)

stop := SHR(size,2)-1;
FOR i := 0 TO stop DO
	PT^[i] := ABS(PT^[i]);
END_FOR;
_ARRAY_ABS := TRUE;


(* revision history
hm	2. apr 2008		rev 1.0
	original version

*)

END_FUNCTION

// oscat_basic/POUs/Mathematical/Array/ARRAY_AVG
FUNCTION ARRAY_AVG : REAL
VAR_INPUT
	pt : POINTER TO ARRAY[0..32000] OF REAL;
	size : UINT;
END_VAR
VAR
	i: UINT;
	stop: UINT;
END_VAR

(*
version 1.3	10. mar. 2009
programmer 	hugo
tested by		tobias

this function will calculate the average of a given array.
the function needs to be called:	array_avg(adr("array"),sizeof("array"));
because this function works with pointers its very time efficient and it needs no extra memory.

*)

stop := SHR(size,2)-1;
ARRAY_AVG := pt^[0];
FOR i := 1 TO stop DO
	ARRAY_AVG := ARRAY_AVG + pt^[i];
END_FOR;
ARRAY_AVG := ARRAY_AVG / UINT_TO_REAL(stop + 1);


(* revision history
hm	2. oct 2007		rev 1.0
	original version

hm	12. dec 2007	rev 1.1
	chaged code for better performance

hm	16. mar. 2008	rev 1.2
	changed input size to uint

hm	10. mar. 2009	rev 1.3
	added type conversion for compatibility reasons
*)

END_FUNCTION

// oscat_basic/POUs/Mathematical/Array/_ARRAY_ADD
FUNCTION _ARRAY_ADD : BOOL
VAR_INPUT
	pt : POINTER TO ARRAY[0..32000] OF REAL;
	size : UINT;
	X : REAL;
END_VAR
VAR
	i: UINT;
	stop: UINT;
END_VAR

(*
version 1.0	2. apr. 2008
programmer 	hugo
tested by	tobias

this function will add an offset X to each element of the array and stroe the result instead of the element.
Array[i] := ARRAY[i] + X.
the function needs to be called:	array_avg(adr("array"),sizeof("array"));
because this function works with pointers its very time efficient and it needs no extra memory.

*)

stop := SHR(size,2)-1;
FOR i := 0 TO stop DO
	PT^[i] := PT^[i] + X;
END_FOR;
_ARRAY_ADD := TRUE;


(* revision history
hm	2. apr 2008		rev 1.0
	original version

*)

END_FUNCTION

// oscat_basic/POUs/Mathematical/Array/_ARRAY_INIT
FUNCTION _ARRAY_INIT : BOOL
VAR_INPUT
	pt : POINTER TO ARRAY[0..32000] OF REAL;
	size : UINT;
	init : REAL;
END_VAR
VAR
	i: UINT;
	stop: UINT;
END_VAR


(*
version 1.3	16 mar 2008
programmer 	hugo
tested by		tobias

this function will initialize a given array with a value init.
the function needs to be called:	_array_init(adr("array"),sizeof("array"));
this function will manipulate a given array.
the function manipulates the original array, it rerturnes true when finished.
because this function works with pointers its very time efficient and it needs no extra memory.

*)

stop := SHR(size,2)-1;
FOR i := 0 TO stop DO
	pt^[i] := init;
END_FOR;

_array_init := TRUE;

(* revision History

hm 6.1.2007		rev 1.1
	change type of function to bool
	added  array_init := true to set output true.

hm	14.11.2007	rev 1.2
	changed stop calculation to be more efficient

hm	16.3. 2008		rev 1.3
	changed type of input size to uint
*)

END_FUNCTION

// oscat_basic/POUs/Mathematical/Array/_ARRAY_MEDIAN
FUNCTION _ARRAY_MEDIAN : REAL
VAR_INPUT
	pt : POINTER TO ARRAY[0..32000] OF REAL;
	size : UINT;
END_VAR
VAR
	i: UINT;
	stop: UINT;
END_VAR

(*
version 1.5	16 mar 2008
programmer 	hugo
tested by		tobias

this function will calculate the median of a given array.
in order to do so the ariginal array is sorted and stays sorted after the function finishes
the function needs to be called:	_array_median(adr("array"),sizeof("array"));
this function will manipulate a given array.
the function will return the median of the original array.
for example [12,0,4,7,1] the median is 4 and the array after the function is called is [0,1,4,7,12]
because this function works with pointers its very time efficient and it needs no extra memory.

*)

_ARRAY_SORT(pt,size);
stop := SHR(size,2)-1;
IF EVEN(UINT_TO_INT(stop)) THEN
	_ARRAY_MEDIAN := pt^[SHR(stop,1)];
ELSE
	i := SHR(stop,1);
	_ARRAY_MEDIAN := (pt^[i] + pt^[i+1]) * 0.5;
END_IF;

(* old code
stop := (size - SIZEOF(pt)) / SIZEOF(pt);
FOR i := 0 TO stop - 1 DO
	FOR m := i + 1 TO stop DO
		IF pt^[i] > pt^[m] THEN
			temp := pt^[i];
			pt^[i] := pt^[m];
			pt^[m] := temp;
		END_IF;
	END_FOR;
END_FOR;
IF even(stop) THEN
	_array_median := pt^[stop/2];
ELSE
	i := stop/2;
	_array_median := (pt^[i] + pt^[i+1])/2;
END_IF;
*)
(* revision history
hm 	3.3.2007		rev 1.1
	corrected an error, changed the statement line 14	i := TRUNC(stop/2); to i := stop/2;

hm		22. sep 2007	rev 1.2
	changed algorithm to use _array_soft for performance reasons

hm		8. oct 2007		rev 1.3
	deleted unused variables m and temp

hm		14. nov 2007	rev 1.4
	corrected a problem with size calculation

hm		16.3. 2008		rev 1.5
	changed type of input size to uint
	performance improvements
*)

END_FUNCTION

// oscat_basic/POUs/Mathematical/Array/_ARRAY_SORT
FUNCTION _ARRAY_SORT : BOOL
VAR_INPUT
	PT : POINTER TO ARRAY[1..32000] OF REAL;
	SIZE : UINT;
END_VAR
VAR
	stack_count: UINT;				(* Laufvariable Stack*)
	stack: ARRAY[1..32] OF UINT;	(* Stackgröße~ 1,6*Log(n)/log(2) *)
										(* Stackgröße 32 => ~1 Mio Elemente *)
	links: UINT;						(* Anfangselement des Arrays *)
	rechts: UINT;						(* Endelement des Arrays *)
	pivot: REAL;						(* temporärer Schwellwert für Tauschbedingung *)
	i: UINT;							(* Laufvariable1 *)
	j: UINT;							(* Laufvariable2 *)
	ende_innen: BOOL;				(* Ende innere Schleife *)
	ende_aussen: BOOL;				(* Ende äußere Schleife *)
	tmp: REAL;						(* Hilfsvariable zum Tauschen von Werten *)
END_VAR



(*
version 2.0	19. jan. 2011
programmer 	Alexander Trikitis
tested by	oscat

this function will sort a given array.
the function needs to be called:	_array_sort(adr("array"),sizeof("array"));
this function will manipulate a given array.
the function will not return anything except true, it will instead manipulate the original array.
because this function works with pointers its very time efficient and it needs no extra memory.

*)

(* Startwerte zur Arraygröße *)
links := 1;					(* Anfangselement des Arrays *)
rechts := SHR(size,2);		(* Endelement des Arrays *)
stack_count := 1;			(* Laufvariable Stack *)

WHILE NOT ende_aussen DO						(* äußere Schleife *)
	IF links < rechts THEN
		pivot := PT^[SHR(rechts+links,1)];			(* Wert des mittleren Elements als Pivot-Wert *)
		i := links -1;
		j := rechts +1;

		(* innere Schleife, teile Feld *)
		ende_innen := FALSE;
		REPEAT

			(* steigende Reihenfolge *)
			REPEAT	i := i+1;	UNTIL (PT^[i] >= pivot) OR NOT (i < rechts)	END_REPEAT;
			REPEAT	j := j-1;	UNTIL (PT^[j] <= pivot) OR NOT (j > links)	END_REPEAT;


			(*sinkende Reihenfolge *)
(*			REPEAT	i := i+1;	UNTIL (PT^[i] <= pivot) OR NOT (i < rechts)	END_REPEAT	*)
(*			REPEAT	j := j-1;	UNTIL (PT^[j] >= pivot) OR NOT (j > links)	END_REPEAT	*)

			IF i >= j THEN
				ende_innen := TRUE;
			ELSE
				   tmp := PT^[j];
				PT^[j] := PT^[i];
				PT^[i] := tmp;
			END_IF;

		UNTIL ende_innen END_REPEAT;

		(* Push stack *)
		stack[stack_count] := rechts;		(* rechten Teil später sortieren *)
		IF Stack_count < 32 THEN
			stack_count := stack_count +1;
		ELSE
			ende_aussen := TRUE;
			_ARRAY_SORT := FALSE;					(* Fehler: Stack zu klein *)
		END_IF;

		(* linken Teil sortiern *)
		rechts := MAX(links, i-1);

	ELSE

		IF stack_count = 1 THEN
			ende_aussen := TRUE;
		ELSE

			links := rechts+1;

			(* pop stack *)
			stack_count := stack_count -1;		(* jetzt rechten Teil sortierne *)
			rechts:= stack[stack_count];
		END_IF;

	END_IF;

END_WHILE;

_ARRAY_SORT := TRUE;				(* Sortierung beendet *)


(* algorithm used before rev 2.0

size := SHR(size,2);
size2 := UINT_TO_INT(SHR(size,1));
FOR i := SIZE2  TO 1 BY -1 DO
	j:=i;
    WHILE j <= SIZE2 DO
     	stop := j * 2 + 1;
        IF stop > UINT_TO_INT(SIZE) THEN stop := stop - 1;
        ELSIF pt^[stop-1] > pt^[stop] THEN stop := stop - 1;
		END_IF;
        IF pt^[j] < pt^[stop] THEN
         	temp := pt^[j];
            pt^[j] := pt^[stop];
            pt^[stop] := temp;
        END_IF;
        j := stop;
    END_WHILE;
END_FOR;

*)

(* heapsort
FOR heapsize := UINT_TO_INT(size) TO 1 BY -1 DO
	popmax := pt^[1];
	pt^[1] := pt^[heapsize];
   	i := 1;
	hs2 := SHR(heapsize,1);
	WHILE i <= hs2 DO
       	stop := i * 2 + 1;  
        	IF stop > heapsize THEN stop := stop - 1;
        	ELSIF pt^[stop-1] > pt^[stop] THEN stop := stop - 1;
	 	END_IF;
        	IF pt^[i] < pt^[stop] THEN
            		temp := pt^[i];
            		pt^[i] := pt^[stop];
            		pt^[stop] := temp;
        	END_IF;
        	i := stop;
    	END_WHILE;
	pt^[heapsize] := popmax;
END_FOR;

_ARRAY_SORT2 := TRUE;
*)

(* old algorithm bubble sort used before rev 1.2
stop := (size - SIZEOF(pt)) / SIZEOF(pt);
FOR i := 0 TO stop - 1 DO
	FOR m := i + 1 TO stop DO
		IF pt^[i] > pt^[m] THEN
			temp := pt^[i];
			pt^[i] := pt^[m];
			pt^[m] := temp;
		END_IF;
	END_FOR;
END_FOR;
_array_sort := TRUE;

*)


(* revision history

hm 	6.1.2007 	rev 1.1
	changed return value to true

hm	22. sep 2007	rev 1.2
	changed sorting algorithm to heap sort for performance reasons

hm 	14. nov 2007	rev 1.3
	changed calculation of stop to be more efficient

hm	15 dec 2007	rev 1.4
	added function return true

hm	5. jan 2008		rev 1.5
	improved performance

hm	16. mar. 2008	rev 1.6
	changed type of input size to uint

hm	28. mar. 2008	rev 1.7
	changed input f to pt

hm	19. jan. 2011	rev 2.0
	new faster algorithm using qucksort (Alexander Drikitis)

*)

END_FUNCTION

// oscat_basic/POUs/Mathematical/Array/_ARRAY_MUL
FUNCTION _ARRAY_MUL : BOOL
VAR_INPUT
	pt : POINTER TO ARRAY[0..32000] OF REAL;
	size : UINT;
	X : REAL;
END_VAR
VAR
	i: UINT;
	stop: UINT;
END_VAR

(*
version 1.0	2. apr. 2008
programmer 	hugo
tested by	tobias

this function will multiply each element of the array and stroe the result instead of the element.
Array[i] := ARRAY[i] * X.
the function needs to be called:	array_avg(adr("array"),sizeof("array"));
because this function works with pointers its very time efficient and it needs no extra memory.

*)

stop := SHR(size,2)-1;
FOR i := 0 TO stop DO
	PT^[i] := PT^[i] * X;
END_FOR;
_ARRAY_MUL := TRUE;


(* revision history
hm	2. apr 2008		rev 1.0
	original version

*)

END_FUNCTION

// oscat_basic/POUs/Mathematical/Array/_ARRAY_SHUFFLE
FUNCTION _ARRAY_SHUFFLE : BOOL
VAR_INPUT
	pt : POINTER TO ARRAY[0..32000] OF REAL;
	size : UINT;
END_VAR
VAR
	temp : REAL;
	pos  : INT;
	i: INT;
	stop: INT;
END_VAR


(*
version 1.2	30. mar. 2008
programmer 	kurt
tested by		hugo

this function will randomly shuffle the elements of an array
*)

stop := UINT_TO_INT(SHR(size,2)-1);
FOR i := 0 TO stop DO
        pos := RDM2(i+pos,0,stop);
        (* swap elements *)
        temp := pt^[i];
        pt^[i] := pt^[pos];
        pt^[pos] := temp;
END_FOR;

_ARRAY_SHUFFLE := TRUE;


(* revision History
hm 	4. mar 2008	rev 1.0
	original version

hm	16. mar. 2008	rev 1.1
	changed type of input size to uint

hm	30. mar. 2008	rev 1.2
	changed last in rdm2 fromm pos to i + pos to allow for more randomness

*)

END_FUNCTION

// oscat_basic/POUs/Mathematical/RDM2
FUNCTION RDM2 : INT
VAR_INPUT
	last : INT;
	low : INT;
	high : INT;
END_VAR


(*
version 1.1	18. oct. 2008
programmer 	hugo
tested by	tobias

this function calculates an integer pseudo random number
the random number will be in the range of low <= rdm2 <= high.

*)

RDM2 := TRUNC_INT(RDM(FRACT(last * math.PI)) * (high - low + 1)) + low;

(* revision history
hm		29. feb 2008		rev 1.0
	original version

hm		18. oct. 2008		rev 1.1
	using math constants

*)

END_FUNCTION

// oscat_basic/POUs/Mathematical/Array/ARRAY_GAV
FUNCTION ARRAY_GAV : REAL
VAR_INPUT
	pt : POINTER TO ARRAY[0..32000] OF REAL;
	size : UINT;
END_VAR
VAR
	i: UINT;
	stop: UINT;
END_VAR

(*
version 1.1	10. mar. 2009
programmer 	hugo
tested by		tobias

this function will calculate the geometric average of a given array.
the function needs to be called:	array_avg(adr("array"),sizeof("array"));
because this function works with pointers its very time efficient and it needs no extra memory.

*)

stop := SHR(size,2)-1;
ARRAY_GAV := 1.0;
FOR i := 0 TO stop DO
	IF pt^[i] > 0.0 THEN
		ARRAY_GAV := ARRAY_GAV * pt^[i];
	ELSE
		ARRAY_GAV := 0.0;
		RETURN;
	END_IF;
END_FOR;
ARRAY_GAV := SQRTN(ARRAY_GAV,UINT_TO_INT(stop)+1);


(* revision history
hm	2. apr 2008	rev 1.0
	original version

hm	10. mar. 2009	rev 1.1
	real constants updated to new systax using dot

*)

END_FUNCTION

// oscat_basic/POUs/Mathematical/SQRTN
FUNCTION SQRTN : REAL
VAR_INPUT
	X : REAL;
	N : INT;
END_VAR


(*
version 1.3	10. mar. 2009
programmer 	hugo
tested by		tobias

this function calculates the nth root function of X according to the formula sqrtn = x^(1/n).

*)

IF N > 0 THEN
	SQRTN := EXP(LN(x) / INT_TO_REAL(n));
ELSE
	SQRTN := 0.0;
END_IF;


(* revision history
hm		12 jan 2007	rev 1.0
	original version

hm		2. dec 2007	rev 1.1
	changed code for better performance

hm		11. mar 2008	rev 1.2
	added result 0 for compatibility reasons

hm 10. mar. 2009	rev 1.3
	added type conversions for compatibility reasons																																																																																																																																																																																																																																																																																																																																																																																																																																																																																																																																																																																																																																																																																																																																																																																																																																																																																																																																																																																																																																																									

*)

END_FUNCTION

// oscat_basic/POUs/Mathematical/Array/ARRAY_HAV
FUNCTION ARRAY_HAV : REAL
VAR_INPUT
	pt : POINTER TO ARRAY[0..32000] OF REAL;
	size : UINT;
END_VAR
VAR
	i: UINT;
	stop: UINT;
END_VAR

(*
version 1.1	10. mar. 2009
programmer 	hugo
tested by		tobias

this function will calculate the harmonic average of a given array.
the function needs to be called:	array_avg(adr("array"),sizeof("array"));
because this function works with pointers its very time efficient and it needs no extra memory.

*)

stop := SHR(size,2)-1;
FOR i := 0 TO stop DO
	IF pt^[i] <> 0.0 THEN
		ARRAY_HAV := ARRAY_HAV + 1.0 / pt^[i];
	ELSE
		ARRAY_HAV := 0.0;
		RETURN;
	END_IF;
END_FOR;
ARRAY_HAV := UINT_TO_REAL(stop + 1) / ARRAY_HAV;


(* revision history
hm	2. apr 2008	rev 1.0
	original version

hm	10. mar. 2009	rev 1.1
	real constants updated to new systax using dot

*)

END_FUNCTION

// oscat_basic/POUs/Mathematical/Array/ARRAY_MAX
FUNCTION ARRAY_MAX : REAL
VAR_INPUT
	pt : POINTER TO ARRAY[0..32000] OF REAL;
	size : UINT;
END_VAR
VAR
	i: UINT;
	stop: UINT;
END_VAR

(*
version 1.1	16. mar. 2008
programmer 	hugo
tested by		tobias

this function will calculate the max value of a given array.
the function needs to be called:	array_max(adr("array"),sizeof("array"));
because this function works with pointers its very time efficient and it needs no extra memory.

*)

stop := (size -SIZEOF(pt)) / SIZEOF(pt);
array_max := pt^[0];
FOR i := 1 TO stop DO
	IF pt^[i] > array_max THEN array_max := pt^[i]; END_IF;
END_FOR;

(* revision history
hm	2. oct 2006		rev 1.0
	original version

hm	16. mar. 2008	rev 1.1
	changed input size to uint
*)

END_FUNCTION

// oscat_basic/POUs/Mathematical/Array/ARRAY_MIN
FUNCTION ARRAY_MIN : REAL
VAR_INPUT
	pt : POINTER TO ARRAY[0..32000] OF REAL;
	size : UINT;
END_VAR
VAR
	i: UINT;
	stop: UINT;
END_VAR

(*
version 1.1	16. mar. 2008
programmer 	hugo
tested by		tobias

this function will calculate the min value of a given array.
the function needs to be called:	array_min(adr("array"),sizeof("array"));
because this function works with pointers its very time efficient and it needs no extra memory.

*)

stop := (size - SIZEOF(pt)) / SIZEOF(pt);
array_min := pt^[0];
FOR i := 1 TO stop DO
	IF pt^[i] < array_min THEN array_min := pt^[i]; END_IF;
END_FOR;


(* revision history
hm		2. oct. 2006
	original version

hm		16. mar. 2008
	changed type of input size to uint

*)

END_FUNCTION

// oscat_basic/POUs/Mathematical/Array/ARRAY_SDV
FUNCTION ARRAY_SDV : REAL
VAR_INPUT
	pt : POINTER TO ARRAY[0..32000] OF REAL;
	size : UINT;
END_VAR


(*
version 1.1	16. mar 2008
programmer 	hugo
tested by		tobias

this function will calculate the standard deviation of a given array.
the function needs to be called:	array_sdv(adr("array"),sizeof("array"));
because this function works with pointers its very time efficient and it needs no extra memory.

*)

(* standard deviation is simply the square root of the variance *)

array_sdv := SQRT(array_var(pt, size));

(* revision history
hm 	1.4.2007		rev 1.0
	function created

hm	16. mar. 2008	rev 1.1
	changed type of input size to uint

*)

END_FUNCTION

// oscat_basic/POUs/Mathematical/Array/ARRAY_VAR
FUNCTION ARRAY_VAR : REAL
VAR_INPUT
	pt : POINTER TO ARRAY[0..32000] OF REAL;
	size : UINT;
END_VAR
VAR
	avg : REAL;
	i: UINT;
	stop: UINT;
END_VAR

(*
version 1.3	10. mar. 2009
programmer 	hugo
tested by		tobias

this function will calculate the variance of a given array.
the function needs to be called:	array_var(adr("array"),sizeof("array"));
because this function works with pointers its very time efficient and it needs no extra memory.

*)

(* at first we calualte the arithmetic average of the array *)

stop := SHR(size,2)-1;
avg := pt^[0];
FOR i := 1 TO stop DO
	avg := avg + pt^[i];
END_FOR;
avg := avg / UINT_TO_REAL(stop + 1);

(* in a second run we calculate the variance of the array *)

array_var := (pt^[0] - avg) * (pt^[0] - avg);
FOR i := 1 TO stop DO
	array_var := array_var + (pt^[i] - avg) * (pt^[i] - avg);
END_FOR;
ARRAY_VAR := ARRAY_VAR / UINT_TO_REAL(stop);

(* revision history
hm 	1.4.2007	rev 1.0
	function created

hm	12.12.2007	rev 1.1
	changed code for better performance

hm	16. mar. 2008	rev 1.2
	changed type of input size to uint

hm	10. mar. 2009	rev 1.3
	added type conversions for compatibility reasons
*)

END_FUNCTION

// oscat_basic/POUs/Mathematical/Array/ARRAY_SPR
FUNCTION ARRAY_SPR : REAL
VAR_INPUT
	pt : POINTER TO ARRAY[0..32000] OF REAL;
	size : UINT;
END_VAR
VAR
	i: UINT;
	stop: UINT;
	array_max : REAL;
	array_min : REAL;
END_VAR

(*
version 1.1	16. mar. 2008
programmer 	hugo
tested by		tobias

this function will calculate the spread of a given array.
the function needs to be called:	array_spr(adr("array"),sizeof("array"));
for example: spread of [12,0,4,1,7] is 12 - 0 = 12.
because this function works with pointers its very time efficient and it needs no extra memory.

*)

stop := (size -SIZEOF(pt)) / SIZEOF(pt);
array_min := pt^[0];
array_max := pt^[0];
FOR i := 1 TO stop DO
	IF pt^[i] > array_max THEN array_max := pt^[i];
	ELSIF pt^[i] < array_min THEN array_min := pt^[i];
	END_IF;
END_FOR;
array_spr := array_max - array_min;


(* revision history
hm 	2. oct. 2006	rev 1.0
	original version

hm	16. mar. 2008	rev 1.1
	changed type of input size to uint

*)

END_FUNCTION

// oscat_basic/POUs/Mathematical/Array/ARRAY_SUM
FUNCTION ARRAY_SUM : REAL
VAR_INPUT
	pt : POINTER TO ARRAY[0..32000] OF REAL;
	size : UINT;
END_VAR
VAR
	i: UINT;
	stop: UINT;
END_VAR


(*
version 1.1	16. mar. 2008
programmer 	hugo
tested by		tobias

this function will calculate the sum of a given array.
the function needs to be called:	array_sum(adr("array"),sizeof("array"));
because this function works with pointers its very time efficient and it needs no extra memory.

*)

stop := (size -SIZEOF(pt)) / SIZEOF(pt);
array_sum := pt^[0];
FOR i := 1 TO stop DO
	array_sum := array_sum + pt^[i];
END_FOR;

(* revision history
hm 	2. oct. 2006	rev 1.0
	function created

hm	16. mar. 2008	rev 1.1
	changed type of input size to uint

*)

END_FUNCTION

// oscat_basic/POUs/Mathematical/Array/ARRAY_TREND
FUNCTION ARRAY_TREND : REAL
VAR_INPUT
	pt : POINTER TO ARRAY[0..32000] OF REAL;
	size : UINT;
END_VAR
VAR
	i: UINT;
	stop: UINT;
	x: REAL;
	stop2: UINT;
END_VAR

(*
version 1.3	10. mar. 2009
programmer 	hugo
tested by		tobias

this function will calculate the trend of a given array.
trend will calculate the avg of the first half of the array and then the avg of the second half, trend = avg2 - avg1.
for example:  [0,1,4,5,3,4,6,3] = 4 - 2.5 = 1.5
the function needs to be called:	array_trend(adr("array"),sizeof("array"));
because this function works with pointers its very time efficient and it needs no extra memory.

*)

stop := SHR(size,2)-1;
stop2 := SHR(stop,1);
FOR i := 0 TO stop2 DO x := x - pt^[i]; END_FOR;
IF EVEN(UINT_TO_INT(stop)) THEN
	FOR i := stop2 TO stop DO X := X + pt^[i]; END_FOR;
ELSE
	FOR i := stop2 + 1 TO stop DO X := X + pt^[i]; END_FOR;
END_IF;
ARRAY_TREND := x / UINT_TO_REAL(stop2 + 1);

(* revision history
hm	2 oct 2007	rev 1.0
	original version

hm	12 dec 2007	rev 1.1
	changed code for better performance

hm	16. mar. 2008	rev 1.2
	changed type of input size to uint

